RoboDK station: Config_1.rdk

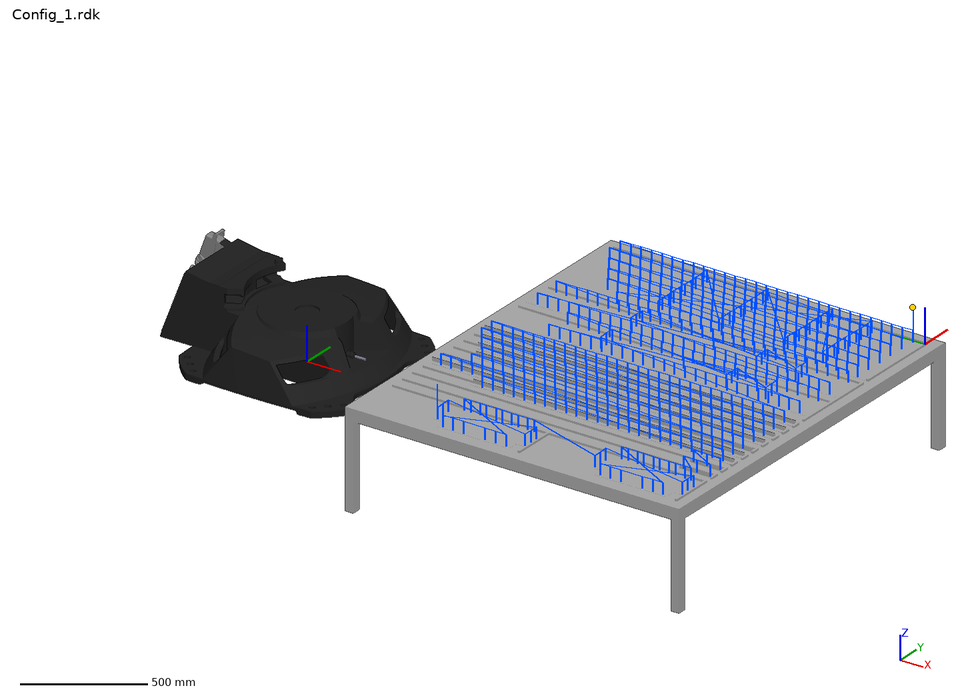
[picture v0: the station drawn from its stored meshes, robots at their saved joint values, targets as dots, program paths as lines]
Station Config_1 (saved by RoboDK 5.2.3). Poses are relative to the parent item; angles as X-Y-Z fixed-axis rotations.
  - frame KUKA KR 210 R2700 extra Base at (0, 0, 0) mm
    - robot KUKA KR 210 R2700 extra: 6 axes, payload 210 kg, reach 2696 mm, repeatability 0.06 mm, weight 1068 kg
        joint limits [-185, -140, -120, -350, -125, -350] to [185, -5, 155, 350, 125, 350]; home [0, -90, 90, 0, 0, 0]; saved at [44.26, -78.74, 122.767, 234.505, 59.006, -215.831]
      - tool Spindle, TCP at (278.6, 0, 88) mm, rotated rx 0 ry 90 rz 0 deg, size 85 x 346.5 x 128 mm
  - frame Corner First Plate at (2495, 660, 510.8) mm, rotated rx 0 ry 0 rz 90 deg
  - object Table 1 at (1700, -800, 455) mm, rotated rx 0 ry 0 rz 90 deg, size 1820 x 1600 x 475 mm, geometry from Table 1.stl
  - object Config_1 at (2495, 660, 510.8) mm, rotated rx 0 ry 0 rz 90 deg
  - machining project Path1 settings: rotZ(0) | rotX(0)*rotY(0) | rotz(0) | onStart | onPathStart | onApproach | onPoint | onRetract | onFinish | SetRPM(%1) | SetTool(%1) | Extruder(%1) | default | default | OutOnMov(%1) | OutOffMov(%1) | onPathFinish | M_RunCode(%1)
  - program Path1 (1740 instructions, listed below)
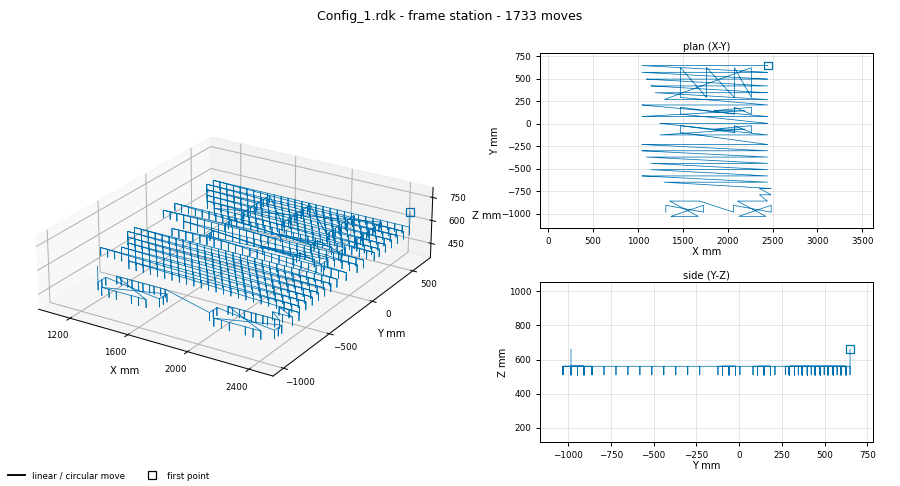
[picture p0: tool path of Config_1.rdk in frame station, 1733 of 1733 moves have a stored position in this frame; points joined in program order, loops and branches not executed]

--- program Path1 (robot KUKA KR 210 R2700 extra) ---
  Smooth(1)
  Set speed (1000.0 mm/s)
  Set Ref.: Corner First Plate
  Set Tool: Spindle
  Show Spindle
  MoveJ 1 to (-10.8, 50, 150) mm, rotated rx 180 ry 0 rz 90 deg; joints [-16.861, -44.669, 69.656, 144.341, 29.838, -148.103]
  MoveL 2 to (-10.8, 50, 150) mm, rotated rx 180 ry 0 rz 90 deg; joints [-16.861, -44.669, 69.656, 144.341, 29.838, -148.103]
  MoveL 3 to (-10.8, 50, 50) mm, rotated rx 180 ry 0 rz 90 deg; joints [-16.861, -42.157, 70.591, 147.522, 32.695, -151.823]
  MoveL 4 to (-10.8, 50, 50) mm, rotated rx 180 ry 0 rz 90 deg; joints [-16.861, -42.157, 70.591, 147.522, 32.695, -151.823]
  Set speed (150.0 mm/s)
  MoveL 5 to (-10.8, 50, -0.5) mm, rotated rx -180 ry 0 rz 90 deg; joints [-16.861, -40.791, 70.897, 148.859, 34.116, -153.424]
  MoveL 6 to (-10.8, 50, 50) mm, rotated rx 180 ry 0 rz 90 deg; joints [-16.861, -42.157, 70.591, 147.522, 32.695, -151.823]
  MoveL 7 to (-10.8, 100, 50) mm, rotated rx -180 ry 0 rz 90 deg; joints [-17.24, -44.27, 74.43, 148.298, 34.333, -152.976]
  MoveL 8 to (-10.8, 100, -0.5) mm, rotated rx -180 ry 0 rz 90 deg; joints [-17.24, -42.862, 74.73, 149.554, 35.795, -154.51]
  MoveL 9 to (-10.8, 100, 50) mm, rotated rx -180 ry 0 rz 90 deg; joints [-17.24, -44.27, 74.43, 148.298, 34.333, -152.976]
  MoveL 10 to (-10.8, 150, 50) mm, rotated rx -180 ry 0 rz 90 deg; joints [-17.637, -46.308, 78.104, 148.894, 35.906, -153.954]
  MoveL 11 to (-10.8, 150, -0.5) mm, rotated rx 180 ry 0 rz 90 deg; joints [-17.637, -44.857, 78.4, 150.085, 37.411, -155.439]
  MoveL 12 to (-10.8, 150, 50) mm, rotated rx -180 ry 0 rz 90 deg; joints [-17.637, -46.308, 78.104, 148.894, 35.906, -153.954]
  MoveL 13 to (-10.8, 200, 50) mm, rotated rx 180 ry 0 rz 90 deg; joints [-18.051, -48.282, 81.634, 149.341, 37.421, -154.79]
  MoveL 14 to (-10.8, 200, -0.5) mm, rotated rx -180 ry 0 rz 90 deg; joints [-18.051, -46.786, 81.927, 150.481, 38.968, -156.24]
  MoveL 15 to (-10.8, 200, 50) mm, rotated rx 180 ry 0 rz 90 deg; joints [-18.051, -48.282, 81.634, 149.341, 37.421, -154.79]
  MoveL 16 to (-10.8, 250, 50) mm, rotated rx 180 ry 0 rz 90 deg; joints [-18.485, -50.201, 85.037, 149.663, 38.882, -155.508]
  MoveL 17 to (-10.8, 250, -0.5) mm, rotated rx -180 ry 0 rz 90 deg; joints [-18.485, -48.66, 85.329, 150.761, 40.473, -156.934]
  MoveL 18 to (-10.8, 250, 50) mm, rotated rx 180 ry 0 rz 90 deg; joints [-18.485, -50.201, 85.037, 149.663, 38.882, -155.508]
  MoveL 19 to (-10.8, 300, 50) mm, rotated rx -180 ry 0 rz 90 deg; joints [-18.939, -52.073, 88.328, 149.877, 40.293, -156.128]
  MoveL 20 to (-10.8, 300, -0.5) mm, rotated rx 180 ry 0 rz 90 deg; joints [-18.939, -50.484, 88.62, 150.941, 41.929, -157.54]
  MoveL 21 to (-10.8, 300, 50) mm, rotated rx -180 ry 0 rz 90 deg; joints [-18.939, -52.073, 88.328, 149.877, 40.293, -156.128]
  MoveL 22 to (-10.8, 350, 50) mm, rotated rx 180 ry 0 rz 90 deg; joints [-19.415, -53.906, 91.518, 149.994, 41.659, -156.663]
  MoveL 23 to (-10.8, 350, -0.5) mm, rotated rx 180 ry 0 rz 90 deg; joints [-19.415, -52.267, 91.81, 151.032, 43.339, -158.069]
  MoveL 24 to (-10.8, 350, 50) mm, rotated rx 180 ry 0 rz 90 deg; joints [-19.415, -53.906, 91.518, 149.994, 41.659, -156.663]
  MoveL 25 to (-10.8, 400, 50) mm, rotated rx 180 ry 0 rz 90 deg; joints [-19.914, -55.704, 94.616, 150.026, 42.981, -157.123]
  MoveL 26 to (-10.8, 400, -0.5) mm, rotated rx -180 ry 0 rz 90 deg; joints [-19.914, -54.013, 94.91, 151.042, 44.709, -158.532]
  MoveL 27 to (-10.8, 400, 50) mm, rotated rx 180 ry 0 rz 90 deg; joints [-19.914, -55.704, 94.616, 150.026, 42.981, -157.123]
  MoveL 28 to (-10.8, 450, 50) mm, rotated rx 180 ry 0 rz 90 deg; joints [-20.439, -57.473, 97.631, 149.977, 44.262, -157.517]
  MoveL 29 to (-10.8, 450, -0.5) mm, rotated rx 180 ry 0 rz 90 deg; joints [-20.439, -55.727, 97.926, 150.978, 46.038, -158.936]
  MoveL 30 to (-10.8, 450, 50) mm, rotated rx 180 ry 0 rz 90 deg; joints [-20.439, -57.473, 97.631, 149.977, 44.262, -157.517]
  MoveL 31 to (-10.8, 500, 50) mm, rotated rx -180 ry 0 rz 90 deg; joints [-20.991, -59.217, 100.569, 149.854, 45.504, -157.852]
  MoveL 32 to (-10.8, 500, -0.5) mm, rotated rx 180 ry 0 rz 90 deg; joints [-20.991, -57.414, 100.867, 150.844, 47.331, -159.288]
  MoveL 33 to (-10.8, 500, 50) mm, rotated rx -180 ry 0 rz 90 deg; joints [-20.991, -59.217, 100.569, 149.854, 45.504, -157.852]
  MoveL 34 to (-10.8, 550, 50) mm, rotated rx 180 ry 0 rz 90 deg; joints [-21.572, -60.942, 103.435, 149.66, 46.709, -158.133]
  MoveL 35 to (-10.8, 550, -0.5) mm, rotated rx 180 ry 0 rz 90 deg; joints [-21.572, -59.078, 103.738, 150.643, 48.588, -159.592]
  MoveL 36 to (-10.8, 550, 50) mm, rotated rx 180 ry 0 rz 90 deg; joints [-21.572, -60.942, 103.435, 149.66, 46.709, -158.133]
  MoveL 37 to (-10.8, 600, 50) mm, rotated rx 180 ry 0 rz 90 deg; joints [-22.185, -62.649, 106.236, 149.397, 47.878, -158.362]
  MoveL 38 to (-10.8, 600, -0.5) mm, rotated rx 180 ry 0 rz 90 deg; joints [-22.185, -60.721, 106.543, 150.377, 49.812, -159.851]
  MoveL 39 to (-10.8, 600, 50) mm, rotated rx 180 ry 0 rz 90 deg; joints [-22.185, -62.649, 106.236, 149.397, 47.878, -158.362]
  MoveL 40 to (-10.8, 650, 50) mm, rotated rx 180 ry 0 rz 90 deg; joints [-22.832, -64.344, 108.975, 149.067, 49.013, -158.542]
  MoveL 41 to (-10.8, 650, -0.5) mm, rotated rx 180 ry 0 rz 90 deg; joints [-22.832, -62.348, 109.287, 150.048, 51.003, -160.069]
  MoveL 42 to (-10.8, 650, 50) mm, rotated rx 180 ry 0 rz 90 deg; joints [-22.832, -64.344, 108.975, 149.067, 49.013, -158.542]
  MoveL 43 to (-10.8, 700, 50) mm, rotated rx -180 ry 0 rz 90 deg; joints [-23.515, -66.029, 111.655, 148.669, 50.113, -158.676]
  MoveL 44 to (-10.8, 700, -0.5) mm, rotated rx 180 ry 0 rz 90 deg; joints [-23.515, -63.961, 111.973, 149.655, 52.163, -160.247]
  MoveL 45 to (-10.8, 700, 50) mm, rotated rx -180 ry 0 rz 90 deg; joints [-23.515, -66.029, 111.655, 148.669, 50.113, -158.676]
  MoveL 46 to (-10.8, 750, 50) mm, rotated rx 180 ry 0 rz 90 deg; joints [-24.238, -67.708, 114.279, 148.204, 51.181, -158.763]
  MoveL 47 to (-10.8, 750, -0.5) mm, rotated rx 180 ry 0 rz 90 deg; joints [-24.238, -65.564, 114.604, 149.198, 53.292, -160.386]
  MoveL 48 to (-10.8, 750, 50) mm, rotated rx 180 ry 0 rz 90 deg; joints [-24.238, -67.708, 114.279, 148.204, 51.181, -158.763]
  MoveL 49 to (-10.8, 800, 50) mm, rotated rx -180 ry 0 rz 90 deg; joints [-25.003, -69.384, 116.85, 147.669, 52.216, -158.805]
  MoveL 50 to (-10.8, 800, -0.5) mm, rotated rx 180 ry 0 rz 90 deg; joints [-25.003, -67.159, 117.183, 148.675, 54.391, -160.488]
  MoveL 51 to (-10.8, 800, 50) mm, rotated rx -180 ry 0 rz 90 deg; joints [-25.003, -69.384, 116.85, 147.669, 52.216, -158.805]
  MoveL 52 to (-10.8, 850, 50) mm, rotated rx -180 ry 0 rz 90 deg; joints [-25.816, -71.061, 119.369, 147.064, 53.22, -158.799]
  MoveL 53 to (-10.8, 850, -0.5) mm, rotated rx 180 ry 0 rz 90 deg; joints [-25.816, -68.749, 119.711, 148.085, 55.46, -160.551]
  MoveL 54 to (-10.8, 850, 50) mm, rotated rx -180 ry 0 rz 90 deg; joints [-25.816, -71.061, 119.369, 147.064, 53.22, -158.799]
  MoveL 55 to (-10.8, 900, 50) mm, rotated rx 180 ry 0 rz 90 deg; joints [-26.678, -72.742, 121.838, 146.383, 54.192, -158.746]
  MoveL 56 to (-10.8, 900, -0.5) mm, rotated rx -180 ry 0 rz 90 deg; joints [-26.678, -70.337, 122.19, 147.424, 56.501, -160.575]
  MoveL 57 to (-10.8, 900, 50) mm, rotated rx 180 ry 0 rz 90 deg; joints [-26.678, -72.742, 121.838, 146.383, 54.192, -158.746]
  MoveL 58 to (-10.8, 950, 50) mm, rotated rx -180 ry 0 rz 90 deg; joints [-27.596, -74.43, 124.259, 145.626, 55.132, -158.641]
  MoveL 59 to (-10.8, 950, -0.5) mm, rotated rx -180 ry 0 rz 90 deg; joints [-27.596, -71.926, 124.621, 146.689, 57.513, -160.559]
  MoveL 60 to (-10.8, 950, 50) mm, rotated rx -180 ry 0 rz 90 deg; joints [-27.596, -74.43, 124.259, 145.626, 55.132, -158.641]
  MoveL 61 to (-10.8, 1000, 50) mm, rotated rx 180 ry 0 rz 90 deg; joints [-28.574, -76.128, 126.631, 144.786, 56.043, -158.484]
  MoveL 62 to (-10.8, 1000, -0.5) mm, rotated rx 180 ry 0 rz 90 deg; joints [-28.574, -73.519, 127.005, 145.877, 58.497, -160.501]
  MoveL 63 to (-10.8, 1000, 50) mm, rotated rx 180 ry 0 rz 90 deg; joints [-28.574, -76.128, 126.631, 144.786, 56.043, -158.484]
  MoveL 64 to (-10.8, 1050, 50) mm, rotated rx -180 ry 0 rz 90 deg; joints [-29.617, -77.842, 128.955, 143.858, 56.923, -158.269]
  MoveL 65 to (-10.8, 1050, -0.5) mm, rotated rx 180 ry 0 rz 90 deg; joints [-29.617, -75.119, 129.342, 144.981, 59.453, -160.398]
  MoveL 66 to (-10.8, 1050, 50) mm, rotated rx -180 ry 0 rz 90 deg; joints [-29.617, -77.842, 128.955, 143.858, 56.923, -158.269]
  MoveL 67 to (-10.8, 1100, 50) mm, rotated rx 180 ry 0 rz 90 deg; joints [-30.732, -79.573, 131.231, 142.838, 57.775, -157.992]
  MoveL 68 to (-10.8, 1100, -0.5) mm, rotated rx -180 ry 0 rz 90 deg; joints [-30.732, -76.729, 131.632, 143.997, 60.382, -160.246]
  MoveL 69 to (-10.8, 1100, 50) mm, rotated rx 180 ry 0 rz 90 deg; joints [-30.732, -79.573, 131.231, 142.838, 57.775, -157.992]
  MoveL 70 to (-10.8, 1150, 50) mm, rotated rx 180 ry 0 rz 90 deg; joints [-31.924, -81.327, 133.457, 141.718, 58.599, -157.647]
  MoveL 71 to (-10.8, 1150, -0.5) mm, rotated rx 180 ry 0 rz 90 deg; joints [-31.924, -78.352, 133.874, 142.918, 61.284, -160.042]
  MoveL 72 to (-10.8, 1150, 50) mm, rotated rx 180 ry 0 rz 90 deg; joints [-31.924, -81.327, 133.457, 141.718, 58.599, -157.647]
  MoveL 73 to (-10.8, 1200, 50) mm, rotated rx 180 ry 0 rz 90 deg; joints [-33.202, -83.108, 135.634, 140.49, 59.397, -157.227]
  MoveL 74 to (-10.8, 1200, -0.5) mm, rotated rx 180 ry 0 rz 90 deg; joints [-33.202, -79.993, 136.068, 141.737, 62.161, -159.78]
  MoveL 75 to (-10.8, 1200, 50) mm, rotated rx 180 ry 0 rz 90 deg; joints [-33.202, -83.108, 135.634, 140.49, 59.397, -157.227]
  MoveL 76 to (-10.8, 1250, 50) mm, rotated rx -180 ry 0 rz 90 deg; joints [-34.574, -84.92, 137.758, 139.147, 60.172, -156.726]
  MoveL 77 to (-10.8, 1250, -0.5) mm, rotated rx -180 ry 0 rz 90 deg; joints [-34.574, -81.654, 138.211, 140.446, 63.014, -159.455]
  MoveL 78 to (-10.8, 1250, 50) mm, rotated rx -180 ry 0 rz 90 deg; joints [-34.574, -84.92, 137.758, 139.147, 60.172, -156.726]
  MoveL 79 to (-10.8, 1300, 50) mm, rotated rx 180 ry 0 rz 90 deg; joints [-36.047, -86.767, 139.828, 137.68, 60.929, -156.133]
  MoveL 80 to (-10.8, 1300, -0.5) mm, rotated rx 180 ry 0 rz 90 deg; joints [-36.047, -83.339, 140.302, 139.037, 63.846, -159.059]
  MoveL 81 to (-10.8, 1300, 50) mm, rotated rx 180 ry 0 rz 90 deg; joints [-36.047, -86.767, 139.828, 137.68, 60.929, -156.133]
  MoveL 82 to (-10.8, 1350, 50) mm, rotated rx 180 ry 0 rz 90 deg; joints [-37.633, -88.655, 141.842, 136.078, 61.671, -155.439]
  MoveL 83 to (-10.8, 1350, -0.5) mm, rotated rx 180 ry 0 rz 90 deg; joints [-37.633, -85.052, 142.339, 137.499, 64.659, -158.585]
  MoveL 84 to (-10.8, 1350, 50) mm, rotated rx 180 ry 0 rz 90 deg; joints [-37.633, -88.655, 141.842, 136.078, 61.671, -155.439]
  MoveL 85 to (-10.8, 1400, 50) mm, rotated rx -180 ry 0 rz 90 deg; joints [-39.341, -90.587, 143.795, 134.333, 62.407, -154.634]
  MoveL 86 to (-10.8, 1400, -0.5) mm, rotated rx 180 ry 0 rz 90 deg; joints [-39.341, -86.798, 144.317, 135.822, 65.461, -158.023]
  MoveL 87 to (-10.8, 1400, 50) mm, rotated rx -180 ry 0 rz 90 deg; joints [-39.341, -90.587, 143.795, 134.333, 62.407, -154.634]
  MoveL 88 to (-10.8, 1450, 50) mm, rotated rx 180 ry 0 rz 90 deg; joints [-41.184, -92.567, 145.684, 132.434, 63.147, -153.707]
  MoveL 89 to (-10.8, 1450, -0.5) mm, rotated rx -180 ry 0 rz 90 deg; joints [-41.184, -88.578, 146.233, 133.998, 66.256, -157.364]
  MoveL 90 to (-10.8, 1450, 50) mm, rotated rx 180 ry 0 rz 90 deg; joints [-41.184, -92.567, 145.684, 132.434, 63.147, -153.707]
  MoveL 91 to (-86.48, 50, 50) mm, rotated rx -180 ry 0 rz 90 deg; joints [-14.989, -43.085, 72.28, 151.237, 32.514, -155.162]
  MoveL 92 to (-86.48, 50, -0.5) mm, rotated rx -180 ry 0 rz 90 deg; joints [-14.989, -41.7, 72.583, 152.451, 34.002, -156.614]
  MoveL 93 to (-86.48, 50, 50) mm, rotated rx -180 ry 0 rz 90 deg; joints [-14.989, -43.085, 72.28, 151.237, 32.514, -155.162]
  MoveL 94 to (-86.48, 100, 50) mm, rotated rx 180 ry 0 rz 90 deg; joints [-15.331, -45.185, 76.083, 151.903, 34.152, -156.164]
  MoveL 95 to (-86.48, 100, -0.5) mm, rotated rx -180 ry 0 rz 90 deg; joints [-15.331, -43.758, 76.381, 153.045, 35.682, -157.556]
  MoveL 96 to (-86.48, 100, 50) mm, rotated rx 180 ry 0 rz 90 deg; joints [-15.331, -45.185, 76.083, 151.903, 34.152, -156.164]
  MoveL 97 to (-86.48, 150, 50) mm, rotated rx 180 ry 0 rz 90 deg; joints [-15.688, -47.215, 79.729, 152.412, 35.724, -157.013]
  MoveL 98 to (-86.48, 150, -0.5) mm, rotated rx 180 ry 0 rz 90 deg; joints [-15.688, -45.744, 80.024, 153.496, 37.296, -158.362]
  MoveL 99 to (-86.48, 150, 50) mm, rotated rx 180 ry 0 rz 90 deg; joints [-15.688, -47.215, 79.729, 152.412, 35.724, -157.013]
  MoveL 100 to (-86.48, 200, 50) mm, rotated rx -180 ry 0 rz 90 deg; joints [-16.062, -49.185, 83.239, 152.79, 37.234, -157.738]
  MoveL 101 to (-86.48, 200, -0.5) mm, rotated rx 180 ry 0 rz 90 deg; joints [-16.062, -47.668, 83.531, 153.829, 38.851, -159.057]
  MoveL 102 to (-86.48, 200, 50) mm, rotated rx -180 ry 0 rz 90 deg; joints [-16.062, -49.185, 83.239, 152.79, 37.234, -157.738]
  MoveL 103 to (-86.48, 250, 50) mm, rotated rx 180 ry 0 rz 90 deg; joints [-16.453, -51.104, 86.628, 153.058, 38.69, -158.361]
  MoveL 104 to (-86.48, 250, -0.5) mm, rotated rx 180 ry 0 rz 90 deg; joints [-16.453, -49.54, 86.92, 154.059, 40.351, -159.659]
  MoveL 105 to (-86.48, 250, 50) mm, rotated rx 180 ry 0 rz 90 deg; joints [-16.453, -51.104, 86.628, 153.058, 38.69, -158.361]
  MoveL 106 to (-86.48, 300, 50) mm, rotated rx -180 ry 0 rz 90 deg; joints [-16.864, -52.98, 89.91, 153.229, 40.094, -158.896]
  MoveL 107 to (-86.48, 300, -0.5) mm, rotated rx 180 ry 0 rz 90 deg; joints [-16.864, -51.367, 90.202, 154.201, 41.802, -160.183]
  MoveL 108 to (-86.48, 300, 50) mm, rotated rx -180 ry 0 rz 90 deg; joints [-16.864, -52.98, 89.91, 153.229, 40.094, -158.896]
  MoveL 109 to (-86.48, 350, 50) mm, rotated rx 180 ry 0 rz 90 deg; joints [-17.294, -54.819, 93.096, 153.315, 41.45, -159.357]
  MoveL 110 to (-86.48, 350, -0.5) mm, rotated rx 180 ry 0 rz 90 deg; joints [-17.294, -53.155, 93.389, 154.264, 43.206, -160.641]
  MoveL 111 to (-86.48, 350, 50) mm, rotated rx 180 ry 0 rz 90 deg; joints [-17.294, -54.819, 93.096, 153.315, 41.45, -159.357]
  MoveL 112 to (-86.48, 400, 50) mm, rotated rx 180 ry 0 rz 90 deg; joints [-17.747, -56.627, 96.194, 153.323, 42.76, -159.751]
  MoveL 113 to (-86.48, 400, -0.5) mm, rotated rx -180 ry 0 rz 90 deg; joints [-17.747, -54.909, 96.489, 154.255, 44.567, -161.039]
  MoveL 114 to (-86.48, 400, 50) mm, rotated rx 180 ry 0 rz 90 deg; joints [-17.747, -56.627, 96.194, 153.323, 42.76, -159.751]
  MoveL 115 to (-86.48, 450, 50) mm, rotated rx 180 ry 0 rz 90 deg; joints [-18.223, -58.41, 99.213, 153.26, 44.028, -160.087]
  MoveL 116 to (-86.48, 450, -0.5) mm, rotated rx -180 ry 0 rz 90 deg; joints [-18.223, -56.634, 99.51, 154.179, 45.887, -161.386]
  MoveL 117 to (-86.48, 450, 50) mm, rotated rx 180 ry 0 rz 90 deg; joints [-18.223, -58.41, 99.213, 153.26, 44.028, -160.087]
  MoveL 118 to (-86.48, 500, 50) mm, rotated rx 180 ry 0 rz 90 deg; joints [-18.725, -60.17, 102.158, 153.129, 45.255, -160.369]
  MoveL 119 to (-86.48, 500, -0.5) mm, rotated rx 180 ry 0 rz 90 deg; joints [-18.725, -58.334, 102.459, 154.04, 47.169, -161.686]
  MoveL 120 to (-86.48, 500, 50) mm, rotated rx 180 ry 0 rz 90 deg; joints [-18.725, -60.17, 102.158, 153.129, 45.255, -160.369]
  MoveL 121 to (-86.48, 550, 50) mm, rotated rx 180 ry 0 rz 90 deg; joints [-19.253, -61.914, 105.035, 152.934, 46.442, -160.602]
  MoveL 122 to (-86.48, 550, -0.5) mm, rotated rx 180 ry 0 rz 90 deg; joints [-19.253, -60.014, 105.341, 153.841, 48.414, -161.943]
  MoveL 123 to (-86.48, 550, 50) mm, rotated rx 180 ry 0 rz 90 deg; joints [-19.253, -61.914, 105.035, 152.934, 46.442, -160.602]
  MoveL 124 to (-86.48, 600, 50) mm, rotated rx 180 ry 0 rz 90 deg; joints [-19.812, -63.645, 107.85, 152.675, 47.591, -160.788]
  MoveL 125 to (-86.48, 600, -0.5) mm, rotated rx 180 ry 0 rz 90 deg; joints [-19.812, -61.677, 108.16, 153.583, 49.623, -162.161]
  MoveL 126 to (-86.48, 600, 50) mm, rotated rx 180 ry 0 rz 90 deg; joints [-19.812, -63.645, 107.85, 152.675, 47.591, -160.788]
  MoveL 127 to (-86.48, 650, 50) mm, rotated rx 180 ry 0 rz 90 deg; joints [-20.402, -65.366, 110.606, 152.354, 48.702, -160.93]
  MoveL 128 to (-86.48, 650, -0.5) mm, rotated rx 180 ry 0 rz 90 deg; joints [-20.402, -63.327, 110.922, 153.265, 50.797, -162.34]
  MoveL 129 to (-86.48, 650, 50) mm, rotated rx 180 ry 0 rz 90 deg; joints [-20.402, -65.366, 110.606, 152.354, 48.702, -160.93]
  MoveL 130 to (-86.48, 700, 50) mm, rotated rx -180 ry 0 rz 90 deg; joints [-21.027, -67.082, 113.306, 151.97, 49.776, -161.027]
  MoveL 131 to (-86.48, 700, -0.5) mm, rotated rx -180 ry 0 rz 90 deg; joints [-21.027, -64.967, 113.629, 152.889, 51.938, -162.482]
  MoveL 132 to (-86.48, 700, 50) mm, rotated rx -180 ry 0 rz 90 deg; joints [-21.027, -67.082, 113.306, 151.97, 49.776, -161.027]
  MoveL 133 to (-86.48, 750, 50) mm, rotated rx -180 ry 0 rz 90 deg; joints [-21.689, -68.796, 115.953, 151.523, 50.813, -161.081]
  MoveL 134 to (-86.48, 750, -0.5) mm, rotated rx 180 ry 0 rz 90 deg; joints [-21.689, -66.6, 116.284, 152.453, 53.044, -162.589]
  MoveL 135 to (-86.48, 750, 50) mm, rotated rx -180 ry 0 rz 90 deg; joints [-21.689, -68.796, 115.953, 151.523, 50.813, -161.081]
  MoveL 136 to (-86.48, 800, 50) mm, rotated rx -180 ry 0 rz 90 deg; joints [-22.392, -70.512, 118.55, 151.01, 51.814, -161.091]
  MoveL 137 to (-86.48, 800, -0.5) mm, rotated rx 180 ry 0 rz 90 deg; joints [-22.392, -68.229, 118.89, 151.955, 54.118, -162.66]
  MoveL 138 to (-86.48, 800, 50) mm, rotated rx -180 ry 0 rz 90 deg; joints [-22.392, -70.512, 118.55, 151.01, 51.814, -161.091]
  MoveL 139 to (-86.48, 850, 50) mm, rotated rx -180 ry 0 rz 90 deg; joints [-23.14, -72.235, 121.099, 150.428, 52.777, -161.056]
  MoveL 140 to (-86.48, 850, -0.5) mm, rotated rx 180 ry 0 rz 90 deg; joints [-23.14, -69.858, 121.448, 151.392, 55.159, -162.694]
  MoveL 141 to (-86.48, 850, 50) mm, rotated rx -180 ry 0 rz 90 deg; joints [-23.14, -72.235, 121.099, 150.428, 52.777, -161.056]
  MoveL 142 to (-86.48, 900, 50) mm, rotated rx 180 ry 0 rz 90 deg; joints [-23.936, -73.967, 123.602, 149.775, 53.704, -160.972]
  MoveL 143 to (-86.48, 900, -0.5) mm, rotated rx 180 ry 0 rz 90 deg; joints [-23.936, -71.491, 123.961, 150.762, 56.166, -162.69]
  MoveL 144 to (-86.48, 900, 50) mm, rotated rx 180 ry 0 rz 90 deg; joints [-23.936, -73.967, 123.602, 149.775, 53.704, -160.972]
  MoveL 145 to (-86.48, 950, 50) mm, rotated rx -180 ry 0 rz 90 deg; joints [-24.786, -75.714, 126.058, 149.045, 54.593, -160.837]
  MoveL 146 to (-86.48, 950, -0.5) mm, rotated rx 180 ry 0 rz 90 deg; joints [-24.786, -73.131, 126.429, 150.06, 57.14, -162.646]
  MoveL 147 to (-86.48, 950, 50) mm, rotated rx -180 ry 0 rz 90 deg; joints [-24.786, -75.714, 126.058, 149.045, 54.593, -160.837]
  MoveL 148 to (-86.48, 1000, 50) mm, rotated rx 180 ry 0 rz 90 deg; joints [-25.694, -77.479, 128.47, 148.234, 55.444, -160.648]
  MoveL 149 to (-86.48, 1000, -0.5) mm, rotated rx 180 ry 0 rz 90 deg; joints [-25.694, -74.781, 128.854, 149.282, 58.079, -162.559]
  MoveL 150 to (-86.48, 1000, 50) mm, rotated rx 180 ry 0 rz 90 deg; joints [-25.694, -77.479, 128.47, 148.234, 55.444, -160.648]
  MoveL 151 to (-86.48, 1050, 50) mm, rotated rx 180 ry 0 rz 90 deg; joints [-26.666, -79.269, 130.836, 147.336, 56.256, -160.398]
  MoveL 152 to (-86.48, 1050, -0.5) mm, rotated rx -180 ry 0 rz 90 deg; joints [-26.666, -76.447, 131.235, 148.422, 58.985, -162.426]
  MoveL 153 to (-86.48, 1050, 50) mm, rotated rx 180 ry 0 rz 90 deg; joints [-26.666, -79.269, 130.836, 147.336, 56.256, -160.398]
  MoveL 154 to (-86.48, 1100, 50) mm, rotated rx 180 ry 0 rz 90 deg; joints [-27.709, -81.088, 133.158, 146.342, 57.029, -160.081]
  MoveL 155 to (-86.48, 1100, -0.5) mm, rotated rx 180 ry 0 rz 90 deg; joints [-27.709, -78.131, 133.573, 147.473, 59.855, -162.242]
  MoveL 156 to (-86.48, 1100, 50) mm, rotated rx 180 ry 0 rz 90 deg; joints [-27.709, -81.088, 133.158, 146.342, 57.029, -160.081]
  MoveL 157 to (-86.48, 1150, 50) mm, rotated rx 180 ry 0 rz 90 deg; joints [-28.829, -82.943, 135.435, 145.246, 57.764, -159.69]
  MoveL 158 to (-86.48, 1150, -0.5) mm, rotated rx 180 ry 0 rz 90 deg; joints [-28.829, -79.841, 135.868, 146.428, 60.689, -162]
  MoveL 159 to (-86.48, 1150, 50) mm, rotated rx 180 ry 0 rz 90 deg; joints [-28.829, -82.943, 135.435, 145.246, 57.764, -159.69]
  MoveL 160 to (-86.48, 1200, 50) mm, rotated rx 180 ry 0 rz 90 deg; joints [-30.034, -84.839, 137.665, 144.036, 58.459, -159.215]
  MoveL 161 to (-86.48, 1200, -0.5) mm, rotated rx -180 ry 0 rz 90 deg; joints [-30.034, -81.58, 138.118, 145.278, 61.487, -161.695]
  MoveL 162 to (-86.48, 1200, 50) mm, rotated rx 180 ry 0 rz 90 deg; joints [-30.034, -84.839, 137.665, 144.036, 58.459, -159.215]
  MoveL 163 to (-86.48, 1250, 50) mm, rotated rx -180 ry 0 rz 90 deg; joints [-31.334, -86.785, 139.848, 142.703, 59.117, -158.645]
  MoveL 164 to (-86.48, 1250, -0.5) mm, rotated rx 180 ry 0 rz 90 deg; joints [-31.334, -83.355, 140.322, 144.012, 62.25, -161.317]
  MoveL 165 to (-86.48, 1250, 50) mm, rotated rx -180 ry 0 rz 90 deg; joints [-31.334, -86.785, 139.848, 142.703, 59.117, -158.645]
  MoveL 166 to (-86.48, 1300, 50) mm, rotated rx -180 ry 0 rz 90 deg; joints [-32.739, -88.788, 141.98, 141.234, 59.738, -157.967]
  MoveL 167 to (-86.48, 1300, -0.5) mm, rotated rx -180 ry 0 rz 90 deg; joints [-32.739, -85.173, 142.478, 142.62, 62.977, -160.857]
  MoveL 168 to (-86.48, 1300, 50) mm, rotated rx -180 ry 0 rz 90 deg; joints [-32.739, -88.788, 141.98, 141.234, 59.738, -157.967]
  MoveL 169 to (-86.48, 1350, 50) mm, rotated rx 180 ry 0 rz 90 deg; joints [-34.26, -90.856, 144.059, 139.615, 60.327, -157.164]
  MoveL 170 to (-86.48, 1350, -0.5) mm, rotated rx -180 ry 0 rz 90 deg; joints [-34.26, -87.04, 144.584, 141.089, 63.67, -160.301]
  MoveL 171 to (-86.48, 1350, 50) mm, rotated rx 180 ry 0 rz 90 deg; joints [-34.26, -90.856, 144.059, 139.615, 60.327, -157.164]
  MoveL 172 to (-86.48, 1400, 50) mm, rotated rx -180 ry 0 rz 90 deg; joints [-35.91, -92.999, 146.082, 137.831, 60.889, -156.219]
  MoveL 173 to (-86.48, 1400, -0.5) mm, rotated rx -180 ry 0 rz 90 deg; joints [-35.91, -88.966, 146.637, 139.404, 64.333, -159.635]
  MoveL 174 to (-86.48, 1400, 50) mm, rotated rx -180 ry 0 rz 90 deg; joints [-35.91, -92.999, 146.082, 137.831, 60.889, -156.219]
  MoveL 175 to (-86.48, 1450, 50) mm, rotated rx 180 ry 0 rz 90 deg; joints [-37.702, -95.228, 148.043, 135.867, 61.433, -155.112]
  MoveL 176 to (-86.48, 1450, -0.5) mm, rotated rx 180 ry 0 rz 90 deg; joints [-37.702, -90.959, 148.632, 137.551, 64.97, -158.843]
  MoveL 177 to (-86.48, 1450, 50) mm, rotated rx 180 ry 0 rz 90 deg; joints [-37.702, -95.228, 148.043, 135.867, 61.433, -155.112]
  MoveL 178 to (-162.16, 50, 50) mm, rotated rx 180 ry 0 rz 90 deg; joints [-13.084, -43.892, 73.746, 154.972, 32.351, -158.474]
  MoveL 179 to (-162.16, 50, -0.5) mm, rotated rx 180 ry 0 rz 90 deg; joints [-13.084, -42.492, 74.047, 156.053, 33.899, -159.764]
  MoveL 180 to (-162.16, 50, 50) mm, rotated rx 180 ry 0 rz 90 deg; joints [-13.084, -43.892, 73.746, 154.972, 32.351, -158.474]
  MoveL 181 to (-162.16, 100, 50) mm, rotated rx 180 ry 0 rz 90 deg; joints [-13.386, -45.983, 77.52, 155.536, 33.989, -159.332]
  MoveL 182 to (-162.16, 100, -0.5) mm, rotated rx 180 ry 0 rz 90 deg; joints [-13.386, -44.539, 77.816, 156.553, 35.579, -160.57]
  MoveL 183 to (-162.16, 100, 50) mm, rotated rx 180 ry 0 rz 90 deg; joints [-13.386, -45.983, 77.52, 155.536, 33.989, -159.332]
  MoveL 184 to (-162.16, 150, 50) mm, rotated rx -180 ry 0 rz 90 deg; joints [-13.701, -48.007, 81.145, 155.964, 35.558, -160.058]
  MoveL 185 to (-162.16, 150, -0.5) mm, rotated rx 180 ry 0 rz 90 deg; joints [-13.701, -46.519, 81.439, 156.931, 37.192, -161.259]
  MoveL 186 to (-162.16, 150, 50) mm, rotated rx -180 ry 0 rz 90 deg; joints [-13.701, -48.007, 81.145, 155.964, 35.558, -160.058]
  MoveL 187 to (-162.16, 200, 50) mm, rotated rx 180 ry 0 rz 90 deg; joints [-14.032, -49.975, 84.639, 156.279, 37.064, -160.678]
  MoveL 188 to (-162.16, 200, -0.5) mm, rotated rx -180 ry 0 rz 90 deg; joints [-14.032, -48.44, 84.931, 157.206, 38.743, -161.852]
  MoveL 189 to (-162.16, 200, 50) mm, rotated rx 180 ry 0 rz 90 deg; joints [-14.032, -49.975, 84.639, 156.279, 37.064, -160.678]
  MoveL 190 to (-162.16, 250, 50) mm, rotated rx 180 ry 0 rz 90 deg; joints [-14.378, -51.896, 88.018, 156.498, 38.514, -161.209]
  MoveL 191 to (-162.16, 250, -0.5) mm, rotated rx 180 ry 0 rz 90 deg; joints [-14.378, -50.312, 88.31, 157.393, 40.239, -162.366]
  MoveL 192 to (-162.16, 250, 50) mm, rotated rx 180 ry 0 rz 90 deg; joints [-14.378, -51.896, 88.018, 156.498, 38.514, -161.209]
  MoveL 193 to (-162.16, 300, 50) mm, rotated rx 180 ry 0 rz 90 deg; joints [-14.742, -53.777, 91.294, 156.633, 39.91, -161.664]
  MoveL 194 to (-162.16, 300, -0.5) mm, rotated rx 180 ry 0 rz 90 deg; joints [-14.742, -52.142, 91.587, 157.503, 41.685, -162.813]
  MoveL 195 to (-162.16, 300, 50) mm, rotated rx 180 ry 0 rz 90 deg; joints [-14.742, -53.777, 91.294, 156.633, 39.91, -161.664]
  MoveL 196 to (-162.16, 350, 50) mm, rotated rx -180 ry 0 rz 90 deg; joints [-15.124, -55.623, 94.478, 156.693, 41.256, -162.054]
  MoveL 197 to (-162.16, 350, -0.5) mm, rotated rx -180 ry 0 rz 90 deg; joints [-15.124, -53.935, 94.772, 157.544, 43.082, -163.202]
  MoveL 198 to (-162.16, 350, 50) mm, rotated rx -180 ry 0 rz 90 deg; joints [-15.124, -55.623, 94.478, 156.693, 41.256, -162.054]
  MoveL 199 to (-162.16, 400, 50) mm, rotated rx 180 ry 0 rz 90 deg; joints [-15.526, -57.442, 97.578, 156.685, 42.556, -162.387]
  MoveL 200 to (-162.16, 400, -0.5) mm, rotated rx 180 ry 0 rz 90 deg; joints [-15.526, -55.697, 97.874, 157.522, 44.436, -163.54]
  MoveL 201 to (-162.16, 400, 50) mm, rotated rx 180 ry 0 rz 90 deg; joints [-15.526, -57.442, 97.578, 156.685, 42.556, -162.387]
  MoveL 202 to (-162.16, 450, 50) mm, rotated rx -180 ry 0 rz 90 deg; joints [-15.949, -59.237, 100.601, 156.614, 43.811, -162.668]
  MoveL 203 to (-162.16, 450, -0.5) mm, rotated rx -180 ry 0 rz 90 deg; joints [-15.949, -57.433, 100.9, 157.441, 45.747, -163.833]
  MoveL 204 to (-162.16, 450, 50) mm, rotated rx -180 ry 0 rz 90 deg; joints [-15.949, -59.237, 100.601, 156.614, 43.811, -162.668]
  MoveL 205 to (-162.16, 500, 50) mm, rotated rx -180 ry 0 rz 90 deg; joints [-16.396, -61.014, 103.555, 156.482, 45.022, -162.902]
  MoveL 206 to (-162.16, 500, -0.5) mm, rotated rx 180 ry 0 rz 90 deg; joints [-16.396, -59.147, 103.858, 157.304, 47.017, -164.085]
  MoveL 207 to (-162.16, 500, 50) mm, rotated rx -180 ry 0 rz 90 deg; joints [-16.396, -61.014, 103.555, 156.482, 45.022, -162.902]
  MoveL 208 to (-162.16, 550, 50) mm, rotated rx -180 ry 0 rz 90 deg; joints [-16.867, -62.777, 106.443, 156.293, 46.192, -163.092]
  MoveL 209 to (-162.16, 550, -0.5) mm, rotated rx 180 ry 0 rz 90 deg; joints [-16.867, -60.844, 106.751, 157.113, 48.25, -164.299]
  MoveL 210 to (-162.16, 550, 50) mm, rotated rx -180 ry 0 rz 90 deg; joints [-16.867, -62.777, 106.443, 156.293, 46.192, -163.092]
  MoveL 211 to (-162.16, 600, 50) mm, rotated rx 180 ry 0 rz 90 deg; joints [-17.365, -64.529, 109.272, 156.047, 47.32, -163.24]
  MoveL 212 to (-162.16, 600, -0.5) mm, rotated rx -180 ry 0 rz 90 deg; joints [-17.365, -62.526, 109.585, 156.869, 49.444, -164.478]
  MoveL 213 to (-162.16, 600, 50) mm, rotated rx 180 ry 0 rz 90 deg; joints [-17.365, -64.529, 109.272, 156.047, 47.32, -163.24]
  MoveL 214 to (-162.16, 650, 50) mm, rotated rx 180 ry 0 rz 90 deg; joints [-17.893, -66.277, 112.044, 155.744, 48.408, -163.347]
  MoveL 215 to (-162.16, 650, -0.5) mm, rotated rx 180 ry 0 rz 90 deg; joints [-17.893, -64.198, 112.364, 156.572, 50.601, -164.622]
  MoveL 216 to (-162.16, 650, 50) mm, rotated rx 180 ry 0 rz 90 deg; joints [-17.893, -66.277, 112.044, 155.744, 48.408, -163.347]
  MoveL 217 to (-162.16, 700, 50) mm, rotated rx 180 ry 0 rz 90 deg; joints [-18.452, -68.022, 114.764, 155.384, 49.455, -163.415]
  MoveL 218 to (-162.16, 700, -0.5) mm, rotated rx 180 ry 0 rz 90 deg; joints [-18.452, -65.863, 115.091, 156.222, 51.722, -164.734]
  MoveL 219 to (-162.16, 700, 50) mm, rotated rx 180 ry 0 rz 90 deg; joints [-18.452, -68.022, 114.764, 155.384, 49.455, -163.415]
  MoveL 220 to (-162.16, 750, 50) mm, rotated rx -180 ry 0 rz 90 deg; joints [-19.047, -69.77, 117.434, 154.965, 50.461, -163.442]
  MoveL 221 to (-162.16, 750, -0.5) mm, rotated rx 180 ry 0 rz 90 deg; joints [-19.047, -67.525, 117.769, 155.816, 52.807, -164.812]
  MoveL 222 to (-162.16, 750, 50) mm, rotated rx -180 ry 0 rz 90 deg; joints [-19.047, -69.77, 117.434, 154.965, 50.461, -163.442]
  MoveL 223 to (-162.16, 800, 50) mm, rotated rx -180 ry 0 rz 90 deg; joints [-19.679, -71.525, 120.057, 154.485, 51.426, -163.427]
  MoveL 224 to (-162.16, 800, -0.5) mm, rotated rx -180 ry 0 rz 90 deg; joints [-19.679, -69.188, 120.401, 155.353, 53.855, -164.857]
  MoveL 225 to (-162.16, 800, 50) mm, rotated rx -180 ry 0 rz 90 deg; joints [-19.679, -71.525, 120.057, 154.485, 51.426, -163.427]
  MoveL 226 to (-162.16, 850, 50) mm, rotated rx -180 ry 0 rz 90 deg; joints [-20.353, -73.292, 122.634, 153.941, 52.348, -163.368]
  MoveL 227 to (-162.16, 850, -0.5) mm, rotated rx 180 ry 0 rz 90 deg; joints [-20.353, -70.855, 122.989, 154.831, 54.865, -164.867]
  MoveL 228 to (-162.16, 850, 50) mm, rotated rx -180 ry 0 rz 90 deg; joints [-20.353, -73.292, 122.634, 153.941, 52.348, -163.368]
  MoveL 229 to (-162.16, 900, 50) mm, rotated rx 180 ry 0 rz 90 deg; joints [-21.073, -75.075, 125.168, 153.328, 53.227, -163.263]
  MoveL 230 to (-162.16, 900, -0.5) mm, rotated rx -180 ry 0 rz 90 deg; joints [-21.073, -72.532, 125.534, 154.244, 55.838, -164.841]
  MoveL 231 to (-162.16, 900, 50) mm, rotated rx 180 ry 0 rz 90 deg; joints [-21.073, -75.075, 125.168, 153.328, 53.227, -163.263]
  MoveL 232 to (-162.16, 950, 50) mm, rotated rx -180 ry 0 rz 90 deg; joints [-21.843, -76.88, 127.659, 152.643, 54.061, -163.108]
  MoveL 233 to (-162.16, 950, -0.5) mm, rotated rx 180 ry 0 rz 90 deg; joints [-21.843, -74.221, 128.038, 153.59, 56.771, -164.776]
  MoveL 234 to (-162.16, 950, 50) mm, rotated rx -180 ry 0 rz 90 deg; joints [-21.843, -76.88, 127.659, 152.643, 54.061, -163.108]
  MoveL 235 to (-162.16, 1000, 50) mm, rotated rx 180 ry 0 rz 90 deg; joints [-22.668, -78.712, 130.108, 151.878, 54.849, -162.897]
  MoveL 236 to (-162.16, 1000, -0.5) mm, rotated rx 180 ry 0 rz 90 deg; joints [-22.668, -75.929, 130.502, 152.863, 57.664, -164.669]
  MoveL 237 to (-162.16, 1000, 50) mm, rotated rx 180 ry 0 rz 90 deg; joints [-22.668, -78.712, 130.108, 151.878, 54.849, -162.897]
  MoveL 238 to (-162.16, 1050, 50) mm, rotated rx -180 ry 0 rz 90 deg; joints [-23.554, -80.578, 132.516, 151.027, 55.587, -162.624]
  MoveL 239 to (-162.16, 1050, -0.5) mm, rotated rx -180 ry 0 rz 90 deg; joints [-23.554, -77.66, 132.926, 152.056, 58.514, -164.514]
  MoveL 240 to (-162.16, 1050, 50) mm, rotated rx -180 ry 0 rz 90 deg; joints [-23.554, -80.578, 132.516, 151.027, 55.587, -162.624]
  MoveL 241 to (-162.16, 1100, 50) mm, rotated rx 180 ry 0 rz 90 deg; joints [-24.508, -82.486, 134.883, 150.082, 56.275, -162.282]
  MoveL 242 to (-162.16, 1100, -0.5) mm, rotated rx 180 ry 0 rz 90 deg; joints [-24.508, -79.42, 135.311, 151.162, 59.319, -164.307]
  MoveL 243 to (-162.16, 1100, 50) mm, rotated rx 180 ry 0 rz 90 deg; joints [-24.508, -82.486, 134.883, 150.082, 56.275, -162.282]
  MoveL 244 to (-162.16, 1150, 50) mm, rotated rx 180 ry 0 rz 90 deg; joints [-25.537, -84.443, 137.208, 149.032, 56.909, -161.859]
  MoveL 245 to (-162.16, 1150, -0.5) mm, rotated rx -180 ry 0 rz 90 deg; joints [-25.537, -81.218, 137.656, 150.172, 60.078, -164.039]
  MoveL 246 to (-162.16, 1150, 50) mm, rotated rx 180 ry 0 rz 90 deg; joints [-25.537, -84.443, 137.208, 149.032, 56.909, -161.859]
  MoveL 247 to (-162.16, 1200, 50) mm, rotated rx 180 ry 0 rz 90 deg; joints [-26.65, -86.46, 139.491, 147.866, 57.487, -161.344]
  MoveL 248 to (-162.16, 1200, -0.5) mm, rotated rx -180 ry 0 rz 90 deg; joints [-26.65, -83.059, 139.961, 149.076, 60.787, -163.702]
  MoveL 249 to (-162.16, 1200, 50) mm, rotated rx 180 ry 0 rz 90 deg; joints [-26.65, -86.46, 139.491, 147.866, 57.487, -161.344]
  MoveL 250 to (-162.16, 1250, 50) mm, rotated rx -180 ry 0 rz 90 deg; joints [-27.856, -88.547, 141.729, 146.569, 58.006, -160.722]
  MoveL 251 to (-162.16, 1250, -0.5) mm, rotated rx -180 ry 0 rz 90 deg; joints [-27.856, -84.954, 142.225, 147.861, 61.443, -163.284]
  MoveL 252 to (-162.16, 1250, 50) mm, rotated rx -180 ry 0 rz 90 deg; joints [-27.856, -88.547, 141.729, 146.569, 58.006, -160.722]
  MoveL 253 to (-162.16, 1300, 50) mm, rotated rx 180 ry 0 rz 90 deg; joints [-29.167, -90.716, 143.922, 145.125, 58.466, -159.973]
  MoveL 254 to (-162.16, 1300, -0.5) mm, rotated rx -180 ry 0 rz 90 deg; joints [-29.167, -86.914, 144.445, 146.514, 62.045, -162.771]
  MoveL 255 to (-162.16, 1300, 50) mm, rotated rx 180 ry 0 rz 90 deg; joints [-29.167, -90.716, 143.922, 145.125, 58.466, -159.973]
  MoveL 256 to (-162.16, 1350, 50) mm, rotated rx 180 ry 0 rz 90 deg; joints [-30.594, -92.982, 146.066, 143.516, 58.866, -159.075]
  MoveL 257 to (-162.16, 1350, -0.5) mm, rotated rx -180 ry 0 rz 90 deg; joints [-30.594, -88.951, 146.621, 145.018, 62.591, -162.145]
  MoveL 258 to (-162.16, 1350, 50) mm, rotated rx 180 ry 0 rz 90 deg; joints [-30.594, -92.982, 146.066, 143.516, 58.866, -159.075]
  MoveL 259 to (-162.16, 1400, 50) mm, rotated rx 180 ry 0 rz 90 deg; joints [-32.153, -95.362, 148.157, 141.719, 59.208, -158.001]
  MoveL 260 to (-162.16, 1400, -0.5) mm, rotated rx 180 ry 0 rz 90 deg; joints [-32.153, -91.079, 148.748, 143.354, 63.078, -161.385]
  MoveL 261 to (-162.16, 1400, 50) mm, rotated rx 180 ry 0 rz 90 deg; joints [-32.153, -95.362, 148.157, 141.719, 59.208, -158.001]
  MoveL 262 to (-237.84, 50, 50) mm, rotated rx 180 ry 0 rz 90 deg; joints [-11.149, -44.582, 74.995, 158.728, 32.207, -161.767]
  MoveL 263 to (-237.84, 50, -0.5) mm, rotated rx -180 ry 0 rz 90 deg; joints [-11.149, -43.168, 75.294, 159.665, 33.809, -162.884]
  MoveL 264 to (-237.84, 50, 50) mm, rotated rx 180 ry 0 rz 90 deg; joints [-11.149, -44.582, 74.995, 158.728, 32.207, -161.767]
  MoveL 265 to (-237.84, 100, 50) mm, rotated rx 180 ry 0 rz 90 deg; joints [-11.409, -46.666, 78.747, 159.196, 33.844, -162.486]
  MoveL 266 to (-237.84, 100, -0.5) mm, rotated rx -180 ry 0 rz 90 deg; joints [-11.409, -45.208, 79.042, 160.078, 35.488, -163.559]
  MoveL 267 to (-237.84, 100, 50) mm, rotated rx 180 ry 0 rz 90 deg; joints [-11.409, -46.666, 78.747, 159.196, 33.844, -162.486]
  MoveL 268 to (-237.84, 150, 50) mm, rotated rx -180 ry 0 rz 90 deg; joints [-11.681, -48.687, 82.355, 159.549, 35.41, -163.094]
  MoveL 269 to (-237.84, 150, -0.5) mm, rotated rx 180 ry 0 rz 90 deg; joints [-11.681, -47.183, 82.648, 160.388, 37.099, -164.135]
  MoveL 270 to (-237.84, 150, 50) mm, rotated rx -180 ry 0 rz 90 deg; joints [-11.681, -48.687, 82.355, 159.549, 35.41, -163.094]
  MoveL 271 to (-237.84, 200, 50) mm, rotated rx 180 ry 0 rz 90 deg; joints [-11.966, -50.655, 85.838, 159.806, 36.912, -163.612]
  MoveL 272 to (-237.84, 200, -0.5) mm, rotated rx 180 ry 0 rz 90 deg; joints [-11.966, -49.103, 86.13, 160.612, 38.647, -164.631]
  MoveL 273 to (-237.84, 200, 50) mm, rotated rx 180 ry 0 rz 90 deg; joints [-11.966, -50.655, 85.838, 159.806, 36.912, -163.612]
  MoveL 274 to (-237.84, 250, 50) mm, rotated rx 180 ry 0 rz 90 deg; joints [-12.264, -52.578, 89.21, 159.982, 38.356, -164.056]
  MoveL 275 to (-237.84, 250, -0.5) mm, rotated rx 180 ry 0 rz 90 deg; joints [-12.264, -50.976, 89.501, 160.761, 40.14, -165.061]
  MoveL 276 to (-237.84, 250, 50) mm, rotated rx 180 ry 0 rz 90 deg; joints [-12.264, -52.578, 89.21, 159.982, 38.356, -164.056]
  MoveL 277 to (-237.84, 300, 50) mm, rotated rx -180 ry 0 rz 90 deg; joints [-12.578, -54.463, 92.482, 160.086, 39.745, -164.435]
  MoveL 278 to (-237.84, 300, -0.5) mm, rotated rx 180 ry 0 rz 90 deg; joints [-12.578, -52.809, 92.775, 160.844, 41.58, -165.434]
  MoveL 279 to (-237.84, 300, 50) mm, rotated rx -180 ry 0 rz 90 deg; joints [-12.578, -54.463, 92.482, 160.086, 39.745, -164.435]
  MoveL 280 to (-237.84, 350, 50) mm, rotated rx 180 ry 0 rz 90 deg; joints [-12.908, -56.317, 95.665, 160.126, 41.082, -164.759]
  MoveL 281 to (-237.84, 350, -0.5) mm, rotated rx 180 ry 0 rz 90 deg; joints [-12.908, -54.608, 95.96, 160.869, 42.971, -165.758]
  MoveL 282 to (-237.84, 350, 50) mm, rotated rx 180 ry 0 rz 90 deg; joints [-12.908, -56.317, 95.665, 160.126, 41.082, -164.759]
  MoveL 283 to (-237.84, 400, 50) mm, rotated rx 180 ry 0 rz 90 deg; joints [-13.256, -58.146, 98.768, 160.108, 42.371, -165.033]
  MoveL 284 to (-237.84, 400, -0.5) mm, rotated rx 180 ry 0 rz 90 deg; joints [-13.256, -56.378, 99.065, 160.839, 44.317, -166.039]
  MoveL 285 to (-237.84, 400, 50) mm, rotated rx 180 ry 0 rz 90 deg; joints [-13.256, -58.146, 98.768, 160.108, 42.371, -165.033]
  MoveL 286 to (-237.84, 450, 50) mm, rotated rx -180 ry 0 rz 90 deg; joints [-13.623, -59.953, 101.797, 160.035, 43.613, -165.264]
  MoveL 287 to (-237.84, 450, -0.5) mm, rotated rx 180 ry 0 rz 90 deg; joints [-13.623, -58.125, 102.097, 160.759, 45.619, -166.281]
  MoveL 288 to (-237.84, 450, 50) mm, rotated rx -180 ry 0 rz 90 deg; joints [-13.623, -59.953, 101.797, 160.035, 43.613, -165.264]
  MoveL 289 to (-237.84, 500, 50) mm, rotated rx -180 ry 0 rz 90 deg; joints [-14.009, -61.745, 104.758, 159.91, 44.81, -165.454]
  MoveL 290 to (-237.84, 500, -0.5) mm, rotated rx 180 ry 0 rz 90 deg; joints [-14.009, -59.852, 105.063, 160.631, 46.879, -166.488]
  MoveL 291 to (-237.84, 500, 50) mm, rotated rx -180 ry 0 rz 90 deg; joints [-14.009, -61.745, 104.758, 159.91, 44.81, -165.454]
  MoveL 292 to (-237.84, 550, 50) mm, rotated rx 180 ry 0 rz 90 deg; joints [-14.419, -63.526, 107.658, 159.734, 45.962, -165.605]
  MoveL 293 to (-237.84, 550, -0.5) mm, rotated rx -180 ry 0 rz 90 deg; joints [-14.419, -61.563, 107.968, 160.455, 48.099, -166.662]
  MoveL 294 to (-237.84, 550, 50) mm, rotated rx 180 ry 0 rz 90 deg; joints [-14.419, -63.526, 107.658, 159.734, 45.962, -165.605]
  MoveL 295 to (-237.84, 600, 50) mm, rotated rx -180 ry 0 rz 90 deg; joints [-14.852, -65.299, 110.5, 159.509, 47.071, -165.72]
  MoveL 296 to (-237.84, 600, -0.5) mm, rotated rx -180 ry 0 rz 90 deg; joints [-14.852, -63.263, 110.816, 160.233, 49.28, -166.806]
  MoveL 297 to (-237.84, 600, 50) mm, rotated rx -180 ry 0 rz 90 deg; joints [-14.852, -65.299, 110.5, 159.509, 47.071, -165.72]
  MoveL 298 to (-237.84, 650, 50) mm, rotated rx -180 ry 0 rz 90 deg; joints [-15.311, -67.071, 113.288, 159.233, 48.136, -165.798]
  MoveL 299 to (-237.84, 650, -0.5) mm, rotated rx -180 ry 0 rz 90 deg; joints [-15.311, -64.956, 113.611, 159.965, 50.421, -166.92]
  MoveL 300 to (-237.84, 650, 50) mm, rotated rx -180 ry 0 rz 90 deg; joints [-15.311, -67.071, 113.288, 159.233, 48.136, -165.798]
  MoveL 301 to (-237.84, 700, 50) mm, rotated rx 180 ry 0 rz 90 deg; joints [-15.799, -68.844, 116.026, 158.906, 49.157, -165.841]
  MoveL 302 to (-237.84, 700, -0.5) mm, rotated rx -180 ry 0 rz 90 deg; joints [-15.799, -66.645, 116.357, 159.649, 51.523, -167.004]
  MoveL 303 to (-237.84, 700, 50) mm, rotated rx 180 ry 0 rz 90 deg; joints [-15.799, -68.844, 116.026, 158.906, 49.157, -165.841]
  MoveL 304 to (-237.84, 750, 50) mm, rotated rx 180 ry 0 rz 90 deg; joints [-16.318, -70.624, 118.717, 158.527, 50.132, -165.848]
  MoveL 305 to (-237.84, 750, -0.5) mm, rotated rx 180 ry 0 rz 90 deg; joints [-16.318, -68.335, 119.057, 159.283, 52.585, -167.059]
  MoveL 306 to (-237.84, 750, 50) mm, rotated rx 180 ry 0 rz 90 deg; joints [-16.318, -70.624, 118.717, 158.527, 50.132, -165.848]
  MoveL 307 to (-237.84, 800, 50) mm, rotated rx -180 ry 0 rz 90 deg; joints [-16.871, -72.415, 121.363, 158.092, 51.062, -165.816]
  MoveL 308 to (-237.84, 800, -0.5) mm, rotated rx -180 ry 0 rz 90 deg; joints [-16.871, -70.029, 121.713, 158.867, 53.608, -167.083]
  MoveL 309 to (-237.84, 800, 50) mm, rotated rx -180 ry 0 rz 90 deg; joints [-16.871, -72.415, 121.363, 158.092, 51.062, -165.816]
  MoveL 310 to (-237.84, 850, 50) mm, rotated rx 180 ry 0 rz 90 deg; joints [-17.462, -74.224, 123.967, 157.598, 51.944, -165.743]
  MoveL 311 to (-237.84, 850, -0.5) mm, rotated rx 180 ry 0 rz 90 deg; joints [-17.462, -71.732, 124.328, 158.396, 54.588, -167.076]
  MoveL 312 to (-237.84, 850, 50) mm, rotated rx 180 ry 0 rz 90 deg; joints [-17.462, -74.224, 123.967, 157.598, 51.944, -165.743]
  MoveL 313 to (-237.84, 900, 50) mm, rotated rx -180 ry 0 rz 90 deg; joints [-18.095, -76.055, 126.529, 157.042, 52.775, -165.627]
  MoveL 314 to (-237.84, 900, -0.5) mm, rotated rx -180 ry 0 rz 90 deg; joints [-18.095, -73.45, 126.903, 157.867, 55.526, -167.035]
  MoveL 315 to (-237.84, 900, 50) mm, rotated rx -180 ry 0 rz 90 deg; joints [-18.095, -76.055, 126.529, 157.042, 52.775, -165.627]
  MoveL 316 to (-237.84, 950, 50) mm, rotated rx -180 ry 0 rz 90 deg; joints [-18.773, -77.915, 129.053, 156.418, 53.554, -165.462]
  MoveL 317 to (-237.84, 950, -0.5) mm, rotated rx -180 ry 0 rz 90 deg; joints [-18.773, -75.187, 129.44, 157.276, 56.418, -166.957]
  MoveL 318 to (-237.84, 950, 50) mm, rotated rx -180 ry 0 rz 90 deg; joints [-18.773, -77.915, 129.053, 156.418, 53.554, -165.462]
  MoveL 319 to (-237.84, 1000, 50) mm, rotated rx 180 ry 0 rz 90 deg; joints [-19.502, -79.811, 131.537, 155.719, 54.276, -165.243]
  MoveL 320 to (-237.84, 1000, -0.5) mm, rotated rx 180 ry 0 rz 90 deg; joints [-19.502, -76.949, 131.94, 156.616, 57.263, -166.839]
  MoveL 321 to (-237.84, 1000, 50) mm, rotated rx 180 ry 0 rz 90 deg; joints [-19.502, -79.811, 131.537, 155.719, 54.276, -165.243]
  MoveL 322 to (-237.84, 1050, 50) mm, rotated rx 180 ry 0 rz 90 deg; joints [-20.288, -81.752, 133.984, 154.937, 54.937, -164.963]
  MoveL 323 to (-237.84, 1050, -0.5) mm, rotated rx -180 ry 0 rz 90 deg; joints [-20.288, -78.744, 134.405, 155.882, 58.055, -166.674]
  MoveL 324 to (-237.84, 1050, 50) mm, rotated rx 180 ry 0 rz 90 deg; joints [-20.288, -81.752, 133.984, 154.937, 54.937, -164.963]
  MoveL 325 to (-237.84, 1100, 50) mm, rotated rx -180 ry 0 rz 90 deg; joints [-21.136, -83.747, 136.392, 154.064, 55.534, -164.611]
  MoveL 326 to (-237.84, 1100, -0.5) mm, rotated rx 180 ry 0 rz 90 deg; joints [-21.136, -80.579, 136.833, 155.065, 58.793, -166.456]
  MoveL 327 to (-237.84, 1100, 50) mm, rotated rx -180 ry 0 rz 90 deg; joints [-21.136, -83.747, 136.392, 154.064, 55.534, -164.611]
  MoveL 328 to (-237.84, 1150, 50) mm, rotated rx 180 ry 0 rz 90 deg; joints [-22.055, -85.806, 138.763, 153.088, 56.06, -164.177]
  MoveL 329 to (-237.84, 1150, -0.5) mm, rotated rx 180 ry 0 rz 90 deg; joints [-22.055, -82.463, 139.226, 154.155, 59.47, -166.176]
  MoveL 330 to (-237.84, 1150, 50) mm, rotated rx 180 ry 0 rz 90 deg; joints [-22.055, -85.806, 138.763, 153.088, 56.06, -164.177]
  MoveL 331 to (-237.84, 1200, 50) mm, rotated rx 180 ry 0 rz 90 deg; joints [-23.053, -87.944, 141.095, 151.996, 56.509, -163.645]
  MoveL 332 to (-237.84, 1200, -0.5) mm, rotated rx 180 ry 0 rz 90 deg; joints [-23.053, -84.408, 141.583, 153.141, 60.081, -165.824]
  MoveL 333 to (-237.84, 1200, 50) mm, rotated rx 180 ry 0 rz 90 deg; joints [-23.053, -87.944, 141.095, 151.996, 56.509, -163.645]
  MoveL 334 to (-237.84, 1250, 50) mm, rotated rx 180 ry 0 rz 90 deg; joints [-24.14, -90.174, 143.388, 150.769, 56.875, -162.997]
  MoveL 335 to (-237.84, 1250, -0.5) mm, rotated rx 180 ry 0 rz 90 deg; joints [-24.14, -86.426, 143.904, 152.009, 60.619, -165.385]
  MoveL 336 to (-237.84, 1250, 50) mm, rotated rx 180 ry 0 rz 90 deg; joints [-24.14, -90.174, 143.388, 150.769, 56.875, -162.997]
  MoveL 337 to (-237.84, 1300, 50) mm, rotated rx 180 ry 0 rz 90 deg; joints [-25.327, -92.517, 145.638, 149.389, 57.15, -162.206]
  MoveL 338 to (-237.84, 1300, -0.5) mm, rotated rx -180 ry 0 rz 90 deg; joints [-25.327, -88.533, 146.186, 150.742, 61.078, -164.841]
  MoveL 339 to (-237.84, 1300, 50) mm, rotated rx 180 ry 0 rz 90 deg; joints [-25.327, -92.517, 145.638, 149.389, 57.15, -162.206]
  MoveL 340 to (-237.84, 1350, 50) mm, rotated rx 180 ry 0 rz 90 deg; joints [-26.628, -94.993, 147.844, 147.829, 57.327, -161.244]
  MoveL 341 to (-237.84, 1350, -0.5) mm, rotated rx 180 ry 0 rz 90 deg; joints [-26.628, -90.749, 148.429, 149.319, 61.448, -164.168]
  MoveL 342 to (-237.84, 1350, 50) mm, rotated rx 180 ry 0 rz 90 deg; joints [-26.628, -94.993, 147.844, 147.829, 57.327, -161.244]
  MoveL 343 to (-313.52, 50, 50) mm, rotated rx 180 ry 0 rz 90 deg; joints [-9.188, -45.157, 76.033, 162.505, 32.084, -165.047]
  MoveL 344 to (-313.52, 50, -0.5) mm, rotated rx -180 ry 0 rz 90 deg; joints [-9.188, -43.731, 76.331, 163.289, 33.732, -165.981]
  MoveL 345 to (-313.52, 50, 50) mm, rotated rx 180 ry 0 rz 90 deg; joints [-9.188, -45.157, 76.033, 162.505, 32.084, -165.047]
  MoveL 346 to (-313.52, 100, 50) mm, rotated rx 180 ry 0 rz 90 deg; joints [-9.404, -47.236, 79.767, 162.882, 33.719, -165.631]
  MoveL 347 to (-313.52, 100, -0.5) mm, rotated rx 180 ry 0 rz 90 deg; joints [-9.404, -45.765, 80.062, 163.621, 35.41, -166.528]
  MoveL 348 to (-313.52, 100, 50) mm, rotated rx 180 ry 0 rz 90 deg; joints [-9.404, -47.236, 79.767, 162.882, 33.719, -165.631]
  MoveL 349 to (-313.52, 150, 50) mm, rotated rx -180 ry 0 rz 90 deg; joints [-9.63, -49.255, 83.363, 163.165, 35.283, -166.126]
  MoveL 350 to (-313.52, 150, -0.5) mm, rotated rx 180 ry 0 rz 90 deg; joints [-9.63, -47.737, 83.656, 163.868, 37.019, -166.996]
  MoveL 351 to (-313.52, 150, 50) mm, rotated rx -180 ry 0 rz 90 deg; joints [-9.63, -49.255, 83.363, 163.165, 35.283, -166.126]
  MoveL 352 to (-313.52, 200, 50) mm, rotated rx 180 ry 0 rz 90 deg; joints [-9.867, -51.223, 86.837, 163.37, 36.781, -166.546]
  MoveL 353 to (-313.52, 200, -0.5) mm, rotated rx -180 ry 0 rz 90 deg; joints [-9.867, -49.656, 87.129, 164.045, 38.565, -167.399]
  MoveL 354 to (-313.52, 200, 50) mm, rotated rx 180 ry 0 rz 90 deg; joints [-9.867, -51.223, 86.837, 163.37, 36.781, -166.546]
  MoveL 355 to (-313.52, 250, 50) mm, rotated rx 180 ry 0 rz 90 deg; joints [-10.116, -53.148, 90.204, 163.507, 38.219, -166.905]
  MoveL 356 to (-313.52, 250, -0.5) mm, rotated rx -180 ry 0 rz 90 deg; joints [-10.116, -51.531, 90.495, 164.16, 40.053, -167.747]
  MoveL 357 to (-313.52, 250, 50) mm, rotated rx 180 ry 0 rz 90 deg; joints [-10.116, -53.148, 90.204, 163.507, 38.219, -166.905]
  MoveL 358 to (-313.52, 300, 50) mm, rotated rx -180 ry 0 rz 90 deg; joints [-10.378, -55.039, 93.474, 163.585, 39.601, -167.211]
  MoveL 359 to (-313.52, 300, -0.5) mm, rotated rx -180 ry 0 rz 90 deg; joints [-10.378, -53.368, 93.767, 164.222, 41.488, -168.049]
  MoveL 360 to (-313.52, 300, 50) mm, rotated rx -180 ry 0 rz 90 deg; joints [-10.378, -55.039, 93.474, 163.585, 39.601, -167.211]
  MoveL 361 to (-313.52, 350, 50) mm, rotated rx 180 ry 0 rz 90 deg; joints [-10.653, -56.9, 96.658, 163.611, 40.931, -167.472]
  MoveL 362 to (-313.52, 350, -0.5) mm, rotated rx 180 ry 0 rz 90 deg; joints [-10.653, -55.172, 96.953, 164.235, 42.874, -168.311]
  MoveL 363 to (-313.52, 350, 50) mm, rotated rx 180 ry 0 rz 90 deg; joints [-10.653, -56.9, 96.658, 163.611, 40.931, -167.472]
  MoveL 364 to (-313.52, 400, 50) mm, rotated rx -180 ry 0 rz 90 deg; joints [-10.943, -58.737, 99.763, 163.587, 42.21, -167.692]
  MoveL 365 to (-313.52, 400, -0.5) mm, rotated rx 180 ry 0 rz 90 deg; joints [-10.943, -56.95, 100.061, 164.203, 44.213, -168.537]
  MoveL 366 to (-313.52, 400, 50) mm, rotated rx -180 ry 0 rz 90 deg; joints [-10.943, -58.737, 99.763, 163.587, 42.21, -167.692]
  MoveL 367 to (-313.52, 450, 50) mm, rotated rx -180 ry 0 rz 90 deg; joints [-11.249, -60.556, 102.798, 163.518, 43.44, -167.876]
  MoveL 368 to (-313.52, 450, -0.5) mm, rotated rx -180 ry 0 rz 90 deg; joints [-11.249, -58.706, 103.1, 164.129, 45.507, -168.731]
  MoveL 369 to (-313.52, 450, 50) mm, rotated rx -180 ry 0 rz 90 deg; joints [-11.249, -60.556, 102.798, 163.518, 43.44, -167.876]
  MoveL 370 to (-313.52, 500, 50) mm, rotated rx -180 ry 0 rz 90 deg; joints [-11.573, -62.362, 105.767, 163.406, 44.623, -168.025]
  MoveL 371 to (-313.52, 500, -0.5) mm, rotated rx 180 ry 0 rz 90 deg; joints [-11.573, -60.445, 106.073, 164.015, 46.758, -168.896]
  MoveL 372 to (-313.52, 500, 50) mm, rotated rx -180 ry 0 rz 90 deg; joints [-11.573, -62.362, 105.767, 163.406, 44.623, -168.025]
  MoveL 373 to (-313.52, 550, 50) mm, rotated rx 180 ry 0 rz 90 deg; joints [-11.915, -64.158, 108.676, 163.251, 45.76, -168.142]
  MoveL 374 to (-313.52, 550, -0.5) mm, rotated rx 180 ry 0 rz 90 deg; joints [-11.915, -62.17, 108.988, 163.861, 47.966, -169.034]
  MoveL 375 to (-313.52, 550, 50) mm, rotated rx 180 ry 0 rz 90 deg; joints [-11.915, -64.158, 108.676, 163.251, 45.76, -168.142]
  MoveL 376 to (-313.52, 600, 50) mm, rotated rx 180 ry 0 rz 90 deg; joints [-12.278, -65.95, 111.53, 163.053, 46.851, -168.228]
  MoveL 377 to (-313.52, 600, -0.5) mm, rotated rx -180 ry 0 rz 90 deg; joints [-12.278, -63.886, 111.849, 163.668, 49.134, -169.146]
  MoveL 378 to (-313.52, 600, 50) mm, rotated rx 180 ry 0 rz 90 deg; joints [-12.278, -65.95, 111.53, 163.053, 46.851, -168.228]
  MoveL 379 to (-313.52, 650, 50) mm, rotated rx -180 ry 0 rz 90 deg; joints [-12.664, -67.743, 114.333, 162.813, 47.894, -168.284]
  MoveL 380 to (-313.52, 650, -0.5) mm, rotated rx 180 ry 0 rz 90 deg; joints [-12.664, -65.597, 114.659, 163.435, 50.26, -169.233]
  MoveL 381 to (-313.52, 650, 50) mm, rotated rx -180 ry 0 rz 90 deg; joints [-12.664, -67.743, 114.333, 162.813, 47.894, -168.284]
  MoveL 382 to (-313.52, 700, 50) mm, rotated rx 180 ry 0 rz 90 deg; joints [-13.074, -69.541, 117.088, 162.529, 48.891, -168.308]
  MoveL 383 to (-313.52, 700, -0.5) mm, rotated rx 180 ry 0 rz 90 deg; joints [-13.074, -67.308, 117.422, 163.162, 51.344, -169.295]
  MoveL 384 to (-313.52, 700, 50) mm, rotated rx 180 ry 0 rz 90 deg; joints [-13.074, -69.541, 117.088, 162.529, 48.891, -168.308]
  MoveL 385 to (-313.52, 750, 50) mm, rotated rx -180 ry 0 rz 90 deg; joints [-13.511, -71.35, 119.797, 162.199, 49.838, -168.301]
  MoveL 386 to (-313.52, 750, -0.5) mm, rotated rx -180 ry 0 rz 90 deg; joints [-13.511, -69.022, 120.141, 162.847, 52.386, -169.331]
  MoveL 387 to (-313.52, 750, 50) mm, rotated rx -180 ry 0 rz 90 deg; joints [-13.511, -71.35, 119.797, 162.199, 49.838, -168.301]
  MoveL 388 to (-313.52, 800, 50) mm, rotated rx 180 ry 0 rz 90 deg; joints [-13.977, -73.174, 122.465, 161.822, 50.734, -168.259]
  MoveL 389 to (-313.52, 800, -0.5) mm, rotated rx -180 ry 0 rz 90 deg; joints [-13.977, -70.745, 122.819, 162.487, 53.384, -169.341]
  MoveL 390 to (-313.52, 800, 50) mm, rotated rx 180 ry 0 rz 90 deg; joints [-13.977, -73.174, 122.465, 161.822, 50.734, -168.259]
  MoveL 391 to (-313.52, 850, 50) mm, rotated rx 180 ry 0 rz 90 deg; joints [-14.477, -75.021, 125.092, 161.392, 51.577, -168.182]
  MoveL 392 to (-313.52, 850, -0.5) mm, rotated rx 180 ry 0 rz 90 deg; joints [-14.477, -72.481, 125.458, 162.08, 54.337, -169.323]
  MoveL 393 to (-313.52, 850, 50) mm, rotated rx 180 ry 0 rz 90 deg; joints [-14.477, -75.021, 125.092, 161.392, 51.577, -168.182]
  MoveL 394 to (-313.52, 900, 50) mm, rotated rx 180 ry 0 rz 90 deg; joints [-15.012, -76.896, 127.68, 160.908, 52.363, -168.065]
  MoveL 395 to (-313.52, 900, -0.5) mm, rotated rx -180 ry 0 rz 90 deg; joints [-15.012, -74.236, 128.06, 161.622, 55.241, -169.275]
  MoveL 396 to (-313.52, 900, 50) mm, rotated rx 180 ry 0 rz 90 deg; joints [-15.012, -76.896, 127.68, 160.908, 52.363, -168.065]
  MoveL 397 to (-313.52, 950, 50) mm, rotated rx -180 ry 0 rz 90 deg; joints [-15.587, -78.807, 130.232, 160.362, 53.087, -167.904]
  MoveL 398 to (-313.52, 950, -0.5) mm, rotated rx -180 ry 0 rz 90 deg; joints [-15.587, -76.017, 130.627, 161.109, 56.094, -169.193]
  MoveL 399 to (-313.52, 950, 50) mm, rotated rx -180 ry 0 rz 90 deg; joints [-15.587, -78.807, 130.232, 160.362, 53.087, -167.904]
  MoveL 400 to (-313.52, 1000, 50) mm, rotated rx 180 ry 0 rz 90 deg; joints [-16.208, -80.762, 132.748, 159.749, 53.745, -167.692]
  MoveL 401 to (-313.52, 1000, -0.5) mm, rotated rx 180 ry 0 rz 90 deg; joints [-16.208, -77.83, 133.16, 160.535, 56.891, -169.073]
  MoveL 402 to (-313.52, 1000, 50) mm, rotated rx 180 ry 0 rz 90 deg; joints [-16.208, -80.762, 132.748, 159.749, 53.745, -167.692]
  MoveL 403 to (-313.52, 1050, 50) mm, rotated rx -180 ry 0 rz 90 deg; joints [-16.878, -82.772, 135.229, 159.061, 54.331, -167.422]
  MoveL 404 to (-313.52, 1050, -0.5) mm, rotated rx -180 ry 0 rz 90 deg; joints [-16.878, -79.684, 135.66, 159.894, 57.627, -168.91]
  MoveL 405 to (-313.52, 1050, 50) mm, rotated rx -180 ry 0 rz 90 deg; joints [-16.878, -82.772, 135.229, 159.061, 54.331, -167.422]
  MoveL 406 to (-313.52, 1100, 50) mm, rotated rx -180 ry 0 rz 90 deg; joints [-17.604, -84.849, 137.676, 158.288, 54.836, -167.084]
  MoveL 407 to (-313.52, 1100, -0.5) mm, rotated rx 180 ry 0 rz 90 deg; joints [-17.604, -81.588, 138.128, 159.177, 58.296, -168.697]
  MoveL 408 to (-313.52, 1100, 50) mm, rotated rx -180 ry 0 rz 90 deg; joints [-17.604, -84.849, 137.676, 158.288, 54.836, -167.084]
  MoveL 409 to (-313.52, 1150, 50) mm, rotated rx 180 ry 0 rz 90 deg; joints [-18.393, -87.005, 140.088, 157.417, 55.251, -166.664]
  MoveL 410 to (-313.52, 1150, -0.5) mm, rotated rx 180 ry 0 rz 90 deg; joints [-18.393, -83.555, 140.565, 158.375, 58.889, -168.424]
  MoveL 411 to (-313.52, 1150, 50) mm, rotated rx 180 ry 0 rz 90 deg; joints [-18.393, -87.005, 140.088, 157.417, 55.251, -166.664]
  MoveL 412 to (-313.52, 1200, 50) mm, rotated rx -180 ry 0 rz 90 deg; joints [-19.253, -89.259, 142.465, 156.435, 55.567, -166.146]
  MoveL 413 to (-313.52, 1200, -0.5) mm, rotated rx -180 ry 0 rz 90 deg; joints [-19.253, -85.599, 142.969, 157.475, 59.399, -168.079]
  MoveL 414 to (-313.52, 1200, 50) mm, rotated rx -180 ry 0 rz 90 deg; joints [-19.253, -89.259, 142.465, 156.435, 55.567, -166.146]
  MoveL 415 to (-313.52, 1250, 50) mm, rotated rx -180 ry 0 rz 90 deg; joints [-20.194, -91.631, 144.806, 155.321, 55.769, -165.507]
  MoveL 416 to (-313.52, 1250, -0.5) mm, rotated rx -180 ry 0 rz 90 deg; joints [-20.194, -87.738, 145.342, 156.462, 59.812, -167.645]
  MoveL 417 to (-313.52, 1250, 50) mm, rotated rx -180 ry 0 rz 90 deg; joints [-20.194, -91.631, 144.806, 155.321, 55.769, -165.507]
  MoveL 418 to (-313.52, 1300, 50) mm, rotated rx -180 ry 0 rz 90 deg; joints [-21.228, -94.146, 147.109, 154.052, 55.843, -164.719]
  MoveL 419 to (-313.52, 1300, -0.5) mm, rotated rx -180 ry 0 rz 90 deg; joints [-21.228, -89.992, 147.681, 155.317, 60.115, -167.102]
  MoveL 420 to (-313.52, 1300, 50) mm, rotated rx -180 ry 0 rz 90 deg; joints [-21.228, -94.146, 147.109, 154.052, 55.843, -164.719]
  MoveL 421 to (-389.2, 50, 50) mm, rotated rx 180 ry 0 rz 90 deg; joints [-7.205, -45.617, 76.862, 166.302, 31.983, -168.319]
  MoveL 422 to (-389.2, 50, -0.5) mm, rotated rx -180 ry 0 rz 90 deg; joints [-7.205, -44.181, 77.159, 166.924, 33.669, -169.06]
  MoveL 423 to (-389.2, 50, 50) mm, rotated rx 180 ry 0 rz 90 deg; joints [-7.205, -45.617, 76.862, 166.302, 31.983, -168.319]
  MoveL 424 to (-389.2, 100, 50) mm, rotated rx 180 ry 0 rz 90 deg; joints [-7.376, -47.693, 80.584, 166.593, 33.617, -168.772]
  MoveL 425 to (-389.2, 100, -0.5) mm, rotated rx 180 ry 0 rz 90 deg; joints [-7.376, -46.211, 80.878, 167.179, 35.346, -169.484]
  MoveL 426 to (-389.2, 100, 50) mm, rotated rx 180 ry 0 rz 90 deg; joints [-7.376, -47.693, 80.584, 166.593, 33.617, -168.772]
  MoveL 427 to (-389.2, 150, 50) mm, rotated rx 180 ry 0 rz 90 deg; joints [-7.554, -49.71, 84.17, 166.81, 35.178, -169.155]
  MoveL 428 to (-389.2, 150, -0.5) mm, rotated rx -180 ry 0 rz 90 deg; joints [-7.554, -48.181, 84.462, 167.368, 36.953, -169.847]
  MoveL 429 to (-389.2, 150, 50) mm, rotated rx 180 ry 0 rz 90 deg; joints [-7.554, -49.71, 84.17, 166.81, 35.178, -169.155]
  MoveL 430 to (-389.2, 200, 50) mm, rotated rx -180 ry 0 rz 90 deg; joints [-7.742, -51.679, 87.638, 166.965, 36.673, -169.481]
  MoveL 431 to (-389.2, 200, -0.5) mm, rotated rx 180 ry 0 rz 90 deg; joints [-7.742, -50.101, 87.93, 167.502, 38.496, -170.158]
  MoveL 432 to (-389.2, 200, 50) mm, rotated rx -180 ry 0 rz 90 deg; joints [-7.742, -51.679, 87.638, 166.965, 36.673, -169.481]
  MoveL 433 to (-389.2, 250, 50) mm, rotated rx -180 ry 0 rz 90 deg; joints [-7.938, -53.608, 91.001, 167.068, 38.106, -169.758]
  MoveL 434 to (-389.2, 250, -0.5) mm, rotated rx 180 ry 0 rz 90 deg; joints [-7.938, -51.977, 91.293, 167.588, 39.982, -170.428]
  MoveL 435 to (-389.2, 250, 50) mm, rotated rx -180 ry 0 rz 90 deg; joints [-7.938, -53.608, 91.001, 167.068, 38.106, -169.758]
  MoveL 436 to (-389.2, 300, 50) mm, rotated rx -180 ry 0 rz 90 deg; joints [-8.145, -55.502, 94.27, 167.125, 39.482, -169.995]
  MoveL 437 to (-389.2, 300, -0.5) mm, rotated rx -180 ry 0 rz 90 deg; joints [-8.145, -53.818, 94.564, 167.632, 41.413, -170.661]
  MoveL 438 to (-389.2, 300, 50) mm, rotated rx -180 ry 0 rz 90 deg; joints [-8.145, -55.502, 94.27, 167.125, 39.482, -169.995]
  MoveL 439 to (-389.2, 350, 50) mm, rotated rx 180 ry 0 rz 90 deg; joints [-8.363, -57.369, 97.455, 167.139, 40.804, -170.195]
  MoveL 440 to (-389.2, 350, -0.5) mm, rotated rx 180 ry 0 rz 90 deg; joints [-8.363, -55.627, 97.751, 167.637, 42.793, -170.863]
  MoveL 441 to (-389.2, 350, 50) mm, rotated rx 180 ry 0 rz 90 deg; joints [-8.363, -57.369, 97.455, 167.139, 40.804, -170.195]
  MoveL 442 to (-389.2, 400, 50) mm, rotated rx 180 ry 0 rz 90 deg; joints [-8.593, -59.215, 100.564, 167.116, 42.075, -170.364]
  MoveL 443 to (-389.2, 400, -0.5) mm, rotated rx 180 ry 0 rz 90 deg; joints [-8.593, -57.412, 100.863, 167.607, 44.126, -171.037]
  MoveL 444 to (-389.2, 400, 50) mm, rotated rx 180 ry 0 rz 90 deg; joints [-8.593, -59.215, 100.564, 167.116, 42.075, -170.364]
  MoveL 445 to (-389.2, 450, 50) mm, rotated rx -180 ry 0 rz 90 deg; joints [-8.836, -61.043, 103.603, 167.056, 43.295, -170.503]
  MoveL 446 to (-389.2, 450, -0.5) mm, rotated rx -180 ry 0 rz 90 deg; joints [-8.836, -59.176, 103.906, 167.544, 45.413, -171.186]
  MoveL 447 to (-389.2, 450, 50) mm, rotated rx -180 ry 0 rz 90 deg; joints [-8.836, -61.043, 103.603, 167.056, 43.295, -170.503]
  MoveL 448 to (-389.2, 500, 50) mm, rotated rx 180 ry 0 rz 90 deg; joints [-9.093, -62.86, 106.579, 166.962, 44.467, -170.616]
  MoveL 449 to (-389.2, 500, -0.5) mm, rotated rx -180 ry 0 rz 90 deg; joints [-9.093, -60.924, 106.887, 167.449, 46.655, -171.312]
  MoveL 450 to (-389.2, 500, 50) mm, rotated rx 180 ry 0 rz 90 deg; joints [-9.093, -62.86, 106.579, 166.962, 44.467, -170.616]
  MoveL 451 to (-389.2, 550, 50) mm, rotated rx -180 ry 0 rz 90 deg; joints [-9.365, -64.67, 109.497, 166.833, 45.59, -170.703]
  MoveL 452 to (-389.2, 550, -0.5) mm, rotated rx 180 ry 0 rz 90 deg; joints [-9.365, -62.661, 109.811, 167.322, 47.855, -171.416]
  MoveL 453 to (-389.2, 550, 50) mm, rotated rx -180 ry 0 rz 90 deg; joints [-9.365, -64.67, 109.497, 166.833, 45.59, -170.703]
  MoveL 454 to (-389.2, 600, 50) mm, rotated rx -180 ry 0 rz 90 deg; joints [-9.654, -66.479, 112.362, 166.67, 46.665, -170.765]
  MoveL 455 to (-389.2, 600, -0.5) mm, rotated rx -180 ry 0 rz 90 deg; joints [-9.654, -64.391, 112.682, 167.164, 49.011, -171.5]
  MoveL 456 to (-389.2, 600, 50) mm, rotated rx -180 ry 0 rz 90 deg; joints [-9.654, -66.479, 112.362, 166.67, 46.665, -170.765]
  MoveL 457 to (-389.2, 650, 50) mm, rotated rx -180 ry 0 rz 90 deg; joints [-9.96, -68.29, 115.177, 166.473, 47.69, -170.802]
  MoveL 458 to (-389.2, 650, -0.5) mm, rotated rx -180 ry 0 rz 90 deg; joints [-9.96, -66.118, 115.505, 166.974, 50.123, -171.563]
  MoveL 459 to (-389.2, 650, 50) mm, rotated rx -180 ry 0 rz 90 deg; joints [-9.96, -68.29, 115.177, 166.473, 47.69, -170.802]
  MoveL 460 to (-389.2, 700, 50) mm, rotated rx 180 ry 0 rz 90 deg; joints [-10.287, -70.109, 117.945, 166.241, 48.665, -170.813]
  MoveL 461 to (-389.2, 700, -0.5) mm, rotated rx 180 ry 0 rz 90 deg; joints [-10.287, -67.847, 118.282, 166.752, 51.192, -171.607]
  MoveL 462 to (-389.2, 700, 50) mm, rotated rx 180 ry 0 rz 90 deg; joints [-10.287, -70.109, 117.945, 166.241, 48.665, -170.813]
  MoveL 463 to (-389.2, 750, 50) mm, rotated rx 180 ry 0 rz 90 deg; joints [-10.636, -71.942, 120.671, 165.971, 49.587, -170.799]
  MoveL 464 to (-389.2, 750, -0.5) mm, rotated rx -180 ry 0 rz 90 deg; joints [-10.636, -69.582, 121.018, 166.495, 52.216, -171.629]
  MoveL 465 to (-389.2, 750, 50) mm, rotated rx 180 ry 0 rz 90 deg; joints [-10.636, -71.942, 120.671, 165.971, 49.587, -170.799]
  MoveL 466 to (-389.2, 800, 50) mm, rotated rx 180 ry 0 rz 90 deg; joints [-11.009, -73.795, 123.356, 165.662, 50.454, -170.756]
  MoveL 467 to (-389.2, 800, -0.5) mm, rotated rx 180 ry 0 rz 90 deg; joints [-11.009, -71.329, 123.714, 166.202, 53.193, -171.63]
  MoveL 468 to (-389.2, 800, 50) mm, rotated rx 180 ry 0 rz 90 deg; joints [-11.009, -73.795, 123.356, 165.662, 50.454, -170.756]
  MoveL 469 to (-389.2, 850, 50) mm, rotated rx -180 ry 0 rz 90 deg; joints [-11.408, -75.674, 126.003, 165.31, 51.262, -170.684]
  MoveL 470 to (-389.2, 850, -0.5) mm, rotated rx 180 ry 0 rz 90 deg; joints [-11.408, -73.093, 126.374, 165.87, 54.12, -171.607]
  MoveL 471 to (-389.2, 850, 50) mm, rotated rx -180 ry 0 rz 90 deg; joints [-11.408, -75.674, 126.003, 165.31, 51.262, -170.684]
  MoveL 472 to (-389.2, 900, 50) mm, rotated rx 180 ry 0 rz 90 deg; joints [-11.838, -77.587, 128.614, 164.912, 52.006, -170.577]
  MoveL 473 to (-389.2, 900, -0.5) mm, rotated rx -180 ry 0 rz 90 deg; joints [-11.838, -74.881, 128.999, 165.496, 54.994, -171.559]
  MoveL 474 to (-389.2, 900, 50) mm, rotated rx 180 ry 0 rz 90 deg; joints [-11.838, -77.587, 128.614, 164.912, 52.006, -170.577]
  MoveL 475 to (-389.2, 950, 50) mm, rotated rx 180 ry 0 rz 90 deg; joints [-12.3, -79.542, 131.19, 164.462, 52.681, -170.432]
  MoveL 476 to (-389.2, 950, -0.5) mm, rotated rx 180 ry 0 rz 90 deg; joints [-12.3, -76.7, 131.591, 165.076, 55.811, -171.482]
  MoveL 477 to (-389.2, 950, 50) mm, rotated rx 180 ry 0 rz 90 deg; joints [-12.3, -79.542, 131.19, 164.462, 52.681, -170.432]
  MoveL 478 to (-389.2, 1000, 50) mm, rotated rx -180 ry 0 rz 90 deg; joints [-12.799, -81.549, 133.733, 163.956, 53.28, -170.244]
  MoveL 479 to (-389.2, 1000, -0.5) mm, rotated rx 180 ry 0 rz 90 deg; joints [-12.799, -78.557, 134.152, 164.605, 56.564, -171.373]
  MoveL 480 to (-389.2, 1000, 50) mm, rotated rx -180 ry 0 rz 90 deg; joints [-12.799, -81.549, 133.733, 163.956, 53.28, -170.244]
  MoveL 481 to (-389.2, 1050, 50) mm, rotated rx 180 ry 0 rz 90 deg; joints [-13.34, -83.621, 136.243, 163.385, 53.795, -170.004]
  MoveL 482 to (-389.2, 1050, -0.5) mm, rotated rx -180 ry 0 rz 90 deg; joints [-13.34, -80.463, 136.683, 164.077, 57.248, -171.226]
  MoveL 483 to (-389.2, 1050, 50) mm, rotated rx 180 ry 0 rz 90 deg; joints [-13.34, -83.621, 136.243, 163.385, 53.795, -170.004]
  MoveL 484 to (-389.2, 1100, 50) mm, rotated rx -180 ry 0 rz 90 deg; joints [-13.928, -85.77, 138.722, 162.74, 54.214, -169.702]
  MoveL 485 to (-389.2, 1100, -0.5) mm, rotated rx -180 ry 0 rz 90 deg; joints [-13.928, -82.43, 139.185, 163.484, 57.852, -171.034]
  MoveL 486 to (-389.2, 1100, 50) mm, rotated rx -180 ry 0 rz 90 deg; joints [-13.928, -85.77, 138.722, 162.74, 54.214, -169.702]
  MoveL 487 to (-389.2, 1150, 50) mm, rotated rx 180 ry 0 rz 90 deg; joints [-14.568, -88.014, 141.17, 162.009, 54.524, -169.327]
  MoveL 488 to (-389.2, 1150, -0.5) mm, rotated rx 180 ry 0 rz 90 deg; joints [-14.568, -84.471, 141.658, 162.817, 58.367, -170.788]
  MoveL 489 to (-389.2, 1150, 50) mm, rotated rx 180 ry 0 rz 90 deg; joints [-14.568, -88.014, 141.17, 162.009, 54.524, -169.327]
  MoveL 490 to (-389.2, 1200, 50) mm, rotated rx -180 ry 0 rz 90 deg; joints [-15.269, -90.374, 143.585, 161.177, 54.709, -168.859]
  MoveL 491 to (-389.2, 1200, -0.5) mm, rotated rx -180 ry 0 rz 90 deg; joints [-15.269, -86.606, 144.104, 162.064, 58.778, -170.476]
  MoveL 492 to (-389.2, 1200, 50) mm, rotated rx -180 ry 0 rz 90 deg; joints [-15.269, -90.374, 143.585, 161.177, 54.709, -168.859]
  MoveL 493 to (-33.64, 230, 50) mm, rotated rx -180 ry 0 rz 90 deg; joints [-17.705, -49.723, 84.193, 150.574, 38.245, -156.107]
  MoveL 494 to (-33.64, 230, -0.5) mm, rotated rx 180 ry 0 rz 90 deg; joints [-17.705, -48.194, 84.485, 151.659, 39.84, -157.503]
  MoveL 495 to (-33.64, 230, 50) mm, rotated rx -180 ry 0 rz 90 deg; joints [-17.705, -49.723, 84.193, 150.574, 38.245, -156.107]
  MoveL 496 to (-63.64, 230, 50) mm, rotated rx 180 ry 0 rz 90 deg; joints [-16.907, -50.081, 84.826, 151.928, 38.17, -157.252]
  MoveL 497 to (-63.64, 230, -0.5) mm, rotated rx 180 ry 0 rz 90 deg; joints [-16.907, -48.543, 85.118, 152.974, 39.792, -158.597]
  MoveL 498 to (-63.64, 230, 50) mm, rotated rx 180 ry 0 rz 90 deg; joints [-16.907, -50.081, 84.826, 151.928, 38.17, -157.252]
  MoveL 499 to (-109.34, 230, 50) mm, rotated rx 180 ry 0 rz 90 deg; joints [-15.677, -50.592, 85.728, 154.003, 38.06, -158.994]
  MoveL 500 to (-109.34, 230, -0.5) mm, rotated rx 180 ry 0 rz 90 deg; joints [-15.677, -49.042, 86.02, 154.986, 39.723, -160.258]
  MoveL 501 to (-109.34, 230, 50) mm, rotated rx 180 ry 0 rz 90 deg; joints [-15.677, -50.592, 85.728, 154.003, 38.06, -158.994]
  MoveL 502 to (-139.34, 230, 50) mm, rotated rx 180 ry 0 rz 90 deg; joints [-14.862, -50.906, 86.281, 155.374, 37.991, -160.137]
  MoveL 503 to (-139.34, 230, -0.5) mm, rotated rx 180 ry 0 rz 90 deg; joints [-14.862, -49.348, 86.572, 156.314, 39.679, -161.344]
  MoveL 504 to (-139.34, 230, 50) mm, rotated rx 180 ry 0 rz 90 deg; joints [-14.862, -50.906, 86.281, 155.374, 37.991, -160.137]
  MoveL 505 to (-185.04, 230, 50) mm, rotated rx 180 ry 0 rz 90 deg; joints [-13.608, -51.351, 87.062, 157.475, 37.891, -161.877]
  MoveL 506 to (-185.04, 230, -0.5) mm, rotated rx -180 ry 0 rz 90 deg; joints [-13.608, -49.781, 87.353, 158.347, 39.616, -162.995]
  MoveL 507 to (-185.04, 230, 50) mm, rotated rx 180 ry 0 rz 90 deg; joints [-13.608, -51.351, 87.062, 157.475, 37.891, -161.877]
  MoveL 508 to (-215.04, 230, 50) mm, rotated rx 180 ry 0 rz 90 deg; joints [-12.778, -51.62, 87.535, 158.862, 37.83, -163.019]
  MoveL 509 to (-215.04, 230, -0.5) mm, rotated rx -180 ry 0 rz 90 deg; joints [-12.778, -50.043, 87.826, 159.687, 39.577, -164.076]
  MoveL 510 to (-215.04, 230, 50) mm, rotated rx 180 ry 0 rz 90 deg; joints [-12.778, -51.62, 87.535, 158.862, 37.83, -163.019]
  MoveL 511 to (-260.74, 230, 50) mm, rotated rx 180 ry 0 rz 90 deg; joints [-11.502, -51.997, 88.196, 160.988, 37.742, -164.758]
  MoveL 512 to (-260.74, 230, -0.5) mm, rotated rx 180 ry 0 rz 90 deg; joints [-11.502, -50.411, 88.487, 161.739, 39.522, -165.72]
  MoveL 513 to (-260.74, 230, 50) mm, rotated rx 180 ry 0 rz 90 deg; joints [-11.502, -51.997, 88.196, 160.988, 37.742, -164.758]
  MoveL 514 to (-290.74, 230, 50) mm, rotated rx 180 ry 0 rz 90 deg; joints [-10.659, -52.223, 88.59, 162.39, 37.689, -165.9]
  MoveL 515 to (-290.74, 230, -0.5) mm, rotated rx 180 ry 0 rz 90 deg; joints [-10.659, -50.631, 88.882, 163.091, 39.488, -166.797]
  MoveL 516 to (-290.74, 230, 50) mm, rotated rx 180 ry 0 rz 90 deg; joints [-10.659, -52.223, 88.59, 162.39, 37.689, -165.9]
  MoveL 517 to (-336.44, 230, 50) mm, rotated rx -180 ry 0 rz 90 deg; joints [-9.365, -52.533, 89.132, 164.538, 37.615, -167.641]
  MoveL 518 to (-336.44, 230, -0.5) mm, rotated rx 180 ry 0 rz 90 deg; joints [-9.365, -50.932, 89.423, 165.16, 39.441, -168.435]
  MoveL 519 to (-336.44, 230, 50) mm, rotated rx -180 ry 0 rz 90 deg; joints [-9.365, -52.533, 89.132, 164.538, 37.615, -167.641]
  MoveL 520 to (-366.44, 230, 50) mm, rotated rx -180 ry 0 rz 90 deg; joints [-8.51, -52.715, 89.448, 165.955, 37.571, -168.785]
  MoveL 521 to (-366.44, 230, -0.5) mm, rotated rx -180 ry 0 rz 90 deg; joints [-8.51, -51.109, 89.74, 166.522, 39.414, -169.51]
  MoveL 522 to (-366.44, 230, 50) mm, rotated rx -180 ry 0 rz 90 deg; joints [-8.51, -52.715, 89.448, 165.955, 37.571, -168.785]
  MoveL 523 to (-33.64, 420, 50) mm, rotated rx -180 ry 0 rz 90 deg; joints [-19.467, -56.706, 96.328, 151.001, 43.429, -158.073]
  MoveL 524 to (-33.64, 420, -0.5) mm, rotated rx -180 ry 0 rz 90 deg; joints [-19.467, -54.985, 96.623, 151.987, 45.2, -159.451]
  MoveL 525 to (-33.64, 420, 50) mm, rotated rx -180 ry 0 rz 90 deg; joints [-19.467, -56.706, 96.328, 151.001, 43.429, -158.073]
  MoveL 526 to (-63.64, 420, 50) mm, rotated rx -180 ry 0 rz 90 deg; joints [-18.6, -57.074, 96.954, 152.306, 43.339, -159.106]
  MoveL 527 to (-63.64, 420, -0.5) mm, rotated rx -180 ry 0 rz 90 deg; joints [-18.6, -55.342, 97.25, 153.258, 45.143, -160.435]
  MoveL 528 to (-63.64, 420, 50) mm, rotated rx -180 ry 0 rz 90 deg; joints [-18.6, -57.074, 96.954, 152.306, 43.339, -159.106]
  MoveL 529 to (-109.34, 420, 50) mm, rotated rx -180 ry 0 rz 90 deg; joints [-17.263, -57.602, 97.85, 154.313, 43.207, -160.681]
  MoveL 530 to (-109.34, 420, -0.5) mm, rotated rx 180 ry 0 rz 90 deg; joints [-17.263, -55.853, 98.146, 155.212, 45.058, -161.933]
  MoveL 531 to (-109.34, 420, 50) mm, rotated rx -180 ry 0 rz 90 deg; joints [-17.263, -57.602, 97.85, 154.313, 43.207, -160.681]
  MoveL 532 to (-139.34, 420, 50) mm, rotated rx 180 ry 0 rz 90 deg; joints [-16.374, -57.927, 98.399, 155.644, 43.124, -161.716]
  MoveL 533 to (-139.34, 420, -0.5) mm, rotated rx 180 ry 0 rz 90 deg; joints [-16.374, -56.167, 98.695, 156.506, 45.004, -162.916]
  MoveL 534 to (-139.34, 420, 50) mm, rotated rx 180 ry 0 rz 90 deg; joints [-16.374, -57.927, 98.399, 155.644, 43.124, -161.716]
  MoveL 535 to (-185.04, 420, 50) mm, rotated rx -180 ry 0 rz 90 deg; joints [-15.005, -58.388, 99.177, 157.692, 43.003, -163.298]
  MoveL 536 to (-185.04, 420, -0.5) mm, rotated rx -180 ry 0 rz 90 deg; joints [-15.005, -56.613, 99.474, 158.493, 44.926, -164.412]
  MoveL 537 to (-185.04, 420, 50) mm, rotated rx -180 ry 0 rz 90 deg; joints [-15.005, -58.388, 99.177, 157.692, 43.003, -163.298]
  MoveL 538 to (-215.04, 420, 50) mm, rotated rx 180 ry 0 rz 90 deg; joints [-14.096, -58.669, 99.649, 159.048, 42.928, -164.338]
  MoveL 539 to (-215.04, 420, -0.5) mm, rotated rx -180 ry 0 rz 90 deg; joints [-14.096, -56.885, 99.947, 159.808, 44.878, -165.394]
  MoveL 540 to (-215.04, 420, 50) mm, rotated rx 180 ry 0 rz 90 deg; joints [-14.096, -58.669, 99.649, 159.048, 42.928, -164.338]
  MoveL 541 to (-260.74, 420, 50) mm, rotated rx -180 ry 0 rz 90 deg; joints [-12.698, -59.063, 100.31, 161.132, 42.821, -165.928]
  MoveL 542 to (-260.74, 420, -0.5) mm, rotated rx 180 ry 0 rz 90 deg; joints [-12.698, -57.265, 100.609, 161.826, 44.808, -166.89]
  MoveL 543 to (-260.74, 420, 50) mm, rotated rx -180 ry 0 rz 90 deg; joints [-12.698, -59.063, 100.31, 161.132, 42.821, -165.928]
  MoveL 544 to (-290.74, 420, 50) mm, rotated rx -180 ry 0 rz 90 deg; joints [-11.771, -59.299, 100.706, 162.512, 42.755, -166.974]
  MoveL 545 to (-290.74, 420, -0.5) mm, rotated rx 180 ry 0 rz 90 deg; joints [-11.771, -57.493, 101.005, 163.161, 44.766, -167.872]
  MoveL 546 to (-290.74, 420, 50) mm, rotated rx -180 ry 0 rz 90 deg; joints [-11.771, -59.299, 100.706, 162.512, 42.755, -166.974]
  MoveL 547 to (-336.44, 420, 50) mm, rotated rx -180 ry 0 rz 90 deg; joints [-10.348, -59.625, 101.249, 164.629, 42.663, -168.572]
  MoveL 548 to (-336.44, 420, -0.5) mm, rotated rx -180 ry 0 rz 90 deg; joints [-10.348, -57.808, 101.549, 165.206, 44.706, -169.369]
  MoveL 549 to (-336.44, 420, 50) mm, rotated rx -180 ry 0 rz 90 deg; joints [-10.348, -59.625, 101.249, 164.629, 42.663, -168.572]
  MoveL 550 to (-366.44, 420, 50) mm, rotated rx -180 ry 0 rz 90 deg; joints [-9.407, -59.815, 101.567, 166.029, 42.608, -169.624]
  MoveL 551 to (-366.44, 420, -0.5) mm, rotated rx -180 ry 0 rz 90 deg; joints [-9.407, -57.992, 101.867, 166.557, 44.671, -170.353]
  MoveL 552 to (-366.44, 420, 50) mm, rotated rx -180 ry 0 rz 90 deg; joints [-9.407, -59.815, 101.567, 166.029, 42.608, -169.624]
  MoveL 553 to (-33.64, 730, 50) mm, rotated rx -180 ry 0 rz 90 deg; joints [-23.192, -67.373, 113.758, 149.385, 50.65, -159.434]
  MoveL 554 to (-33.64, 730, -0.5) mm, rotated rx 180 ry 0 rz 90 deg; joints [-23.192, -65.244, 114.082, 150.357, 52.771, -161.002]
  MoveL 555 to (-33.64, 730, 50) mm, rotated rx -180 ry 0 rz 90 deg; joints [-23.192, -67.373, 113.758, 149.385, 50.65, -159.434]
  MoveL 556 to (-63.64, 730, 50) mm, rotated rx 180 ry 0 rz 90 deg; joints [-22.191, -67.798, 114.418, 150.698, 50.509, -160.358]
  MoveL 557 to (-63.64, 730, -0.5) mm, rotated rx 180 ry 0 rz 90 deg; joints [-22.191, -65.65, 114.744, 151.644, 52.677, -161.88]
  MoveL 558 to (-63.64, 730, 50) mm, rotated rx 180 ry 0 rz 90 deg; joints [-22.191, -67.798, 114.418, 150.698, 50.509, -160.358]
  MoveL 559 to (-109.34, 730, 50) mm, rotated rx -180 ry 0 rz 90 deg; joints [-20.639, -68.413, 115.366, 152.734, 50.298, -161.777]
  MoveL 560 to (-109.34, 730, -0.5) mm, rotated rx 180 ry 0 rz 90 deg; joints [-20.639, -66.235, 115.694, 153.636, 52.535, -163.223]
  MoveL 561 to (-109.34, 730, 50) mm, rotated rx -180 ry 0 rz 90 deg; joints [-20.639, -68.413, 115.366, 152.734, 50.298, -161.777]
  MoveL 562 to (-139.34, 730, 50) mm, rotated rx 180 ry 0 rz 90 deg; joints [-19.602, -68.793, 115.949, 154.093, 50.163, -162.716]
  MoveL 563 to (-139.34, 730, -0.5) mm, rotated rx 180 ry 0 rz 90 deg; joints [-19.602, -66.597, 116.279, 154.964, 52.445, -164.109]
  MoveL 564 to (-139.34, 730, 50) mm, rotated rx 180 ry 0 rz 90 deg; joints [-19.602, -68.793, 115.949, 154.093, 50.163, -162.716]
  MoveL 565 to (-185.04, 730, 50) mm, rotated rx -180 ry 0 rz 90 deg; joints [-17.997, -69.337, 116.778, 156.2, 49.965, -164.161]
  MoveL 566 to (-185.04, 730, -0.5) mm, rotated rx -180 ry 0 rz 90 deg; joints [-17.997, -67.114, 117.111, 157.018, 52.311, -165.464]
  MoveL 567 to (-185.04, 730, 50) mm, rotated rx -180 ry 0 rz 90 deg; joints [-17.997, -69.337, 116.778, 156.2, 49.965, -164.161]
  MoveL 568 to (-215.04, 730, 50) mm, rotated rx -180 ry 0 rz 90 deg; joints [-16.928, -69.671, 117.283, 157.605, 49.84, -165.118]
  MoveL 569 to (-215.04, 730, -0.5) mm, rotated rx -180 ry 0 rz 90 deg; joints [-16.928, -67.43, 117.618, 158.386, 52.227, -166.358]
  MoveL 570 to (-215.04, 730, 50) mm, rotated rx -180 ry 0 rz 90 deg; joints [-16.928, -69.671, 117.283, 157.605, 49.84, -165.118]
  MoveL 571 to (-260.74, 730, 50) mm, rotated rx -180 ry 0 rz 90 deg; joints [-15.275, -70.14, 117.992, 159.779, 49.658, -166.589]
  MoveL 572 to (-260.74, 730, -0.5) mm, rotated rx 180 ry 0 rz 90 deg; joints [-15.275, -67.876, 118.329, 160.498, 52.105, -167.728]
  MoveL 573 to (-260.74, 730, 50) mm, rotated rx -180 ry 0 rz 90 deg; joints [-15.275, -70.14, 117.992, 159.779, 49.658, -166.589]
  MoveL 574 to (-290.74, 730, 50) mm, rotated rx 180 ry 0 rz 90 deg; joints [-14.175, -70.424, 118.417, 161.227, 49.546, -167.563]
  MoveL 575 to (-290.74, 730, -0.5) mm, rotated rx 180 ry 0 rz 90 deg; joints [-14.175, -68.145, 118.756, 161.902, 52.029, -168.631]
  MoveL 576 to (-290.74, 730, 50) mm, rotated rx 180 ry 0 rz 90 deg; joints [-14.175, -70.424, 118.417, 161.227, 49.546, -167.563]
  MoveL 577 to (-336.44, 730, 50) mm, rotated rx 180 ry 0 rz 90 deg; joints [-12.479, -70.815, 119.003, 163.462, 49.387, -169.06]
  MoveL 578 to (-336.44, 730, -0.5) mm, rotated rx -180 ry 0 rz 90 deg; joints [-12.479, -68.516, 119.344, 164.067, 51.922, -170.015]
  MoveL 579 to (-336.44, 730, 50) mm, rotated rx 180 ry 0 rz 90 deg; joints [-12.479, -70.815, 119.003, 163.462, 49.387, -169.06]
  MoveL 580 to (-366.44, 730, 50) mm, rotated rx 180 ry 0 rz 90 deg; joints [-11.354, -71.046, 119.347, 164.948, 49.292, -170.052]
  MoveL 581 to (-366.44, 730, -0.5) mm, rotated rx 180 ry 0 rz 90 deg; joints [-11.354, -68.735, 119.689, 165.504, 51.858, -170.928]
  MoveL 582 to (-366.44, 730, 50) mm, rotated rx 180 ry 0 rz 90 deg; joints [-11.354, -71.046, 119.347, 164.948, 49.292, -170.052]
  MoveL 583 to (-33.64, 1020, 50) mm, rotated rx 180 ry 0 rz 90 deg; joints [-28.122, -77.24, 128.147, 145.449, 56.211, -159.045]
  MoveL 584 to (-33.64, 1020, -0.5) mm, rotated rx -180 ry 0 rz 90 deg; joints [-28.122, -74.558, 128.529, 146.542, 58.751, -161.078]
  MoveL 585 to (-33.64, 1020, 50) mm, rotated rx 180 ry 0 rz 90 deg; joints [-28.122, -77.24, 128.147, 145.449, 56.211, -159.045]
  MoveL 586 to (-63.64, 1020, 50) mm, rotated rx -180 ry 0 rz 90 deg; joints [-26.969, -77.787, 128.882, 146.82, 55.963, -159.897]
  MoveL 587 to (-63.64, 1020, -0.5) mm, rotated rx -180 ry 0 rz 90 deg; joints [-26.969, -75.068, 129.269, 147.897, 58.578, -161.889]
  MoveL 588 to (-63.64, 1020, 50) mm, rotated rx -180 ry 0 rz 90 deg; joints [-26.969, -77.787, 128.882, 146.82, 55.963, -159.897]
  MoveL 589 to (-109.34, 1020, 50) mm, rotated rx 180 ry 0 rz 90 deg; joints [-25.166, -78.587, 129.943, 148.971, 55.584, -161.222]
  MoveL 590 to (-109.34, 1020, -0.5) mm, rotated rx -180 ry 0 rz 90 deg; joints [-25.166, -75.812, 130.336, 150.017, 58.313, -163.14]
  MoveL 591 to (-109.34, 1020, 50) mm, rotated rx 180 ry 0 rz 90 deg; joints [-25.166, -78.587, 129.943, 148.971, 55.584, -161.222]
  MoveL 592 to (-139.34, 1020, 50) mm, rotated rx 180 ry 0 rz 90 deg; joints [-23.953, -79.087, 130.599, 150.423, 55.337, -162.11]
  MoveL 593 to (-139.34, 1020, -0.5) mm, rotated rx -180 ry 0 rz 90 deg; joints [-23.953, -76.277, 130.996, 151.445, 58.14, -163.973]
  MoveL 594 to (-139.34, 1020, 50) mm, rotated rx 180 ry 0 rz 90 deg; joints [-23.953, -79.087, 130.599, 150.423, 55.337, -162.11]
  MoveL 595 to (-185.04, 1020, 50) mm, rotated rx 180 ry 0 rz 90 deg; joints [-22.061, -79.81, 131.535, 152.697, 54.965, -163.493]
  MoveL 596 to (-185.04, 1020, -0.5) mm, rotated rx -180 ry 0 rz 90 deg; joints [-22.061, -76.948, 131.939, 153.675, 57.879, -165.261]
  MoveL 597 to (-185.04, 1020, 50) mm, rotated rx 180 ry 0 rz 90 deg; joints [-22.061, -79.81, 131.535, 152.697, 54.965, -163.493]
  MoveL 598 to (-215.04, 1020, 50) mm, rotated rx -180 ry 0 rz 90 deg; joints [-20.79, -80.257, 132.108, 154.23, 54.726, -164.422]
  MoveL 599 to (-215.04, 1020, -0.5) mm, rotated rx -180 ry 0 rz 90 deg; joints [-20.79, -77.362, 132.515, 155.174, 57.711, -166.119]
  MoveL 600 to (-215.04, 1020, 50) mm, rotated rx -180 ry 0 rz 90 deg; joints [-20.79, -80.257, 132.108, 154.23, 54.726, -164.422]
  MoveL 601 to (-260.74, 1020, 50) mm, rotated rx 180 ry 0 rz 90 deg; joints [-18.812, -80.894, 132.914, 156.626, 54.373, -165.869]
  MoveL 602 to (-260.74, 1020, -0.5) mm, rotated rx -180 ry 0 rz 90 deg; joints [-18.812, -77.952, 133.327, 157.511, 57.463, -167.447]
  MoveL 603 to (-260.74, 1020, 50) mm, rotated rx 180 ry 0 rz 90 deg; joints [-18.812, -80.894, 132.914, 156.626, 54.373, -165.869]
  MoveL 604 to (-290.74, 1020, 50) mm, rotated rx -180 ry 0 rz 90 deg; joints [-17.488, -81.282, 133.4, 158.239, 54.151, -166.842]
  MoveL 605 to (-290.74, 1020, -0.5) mm, rotated rx 180 ry 0 rz 90 deg; joints [-17.488, -78.31, 133.816, 159.079, 57.307, -168.333]
  MoveL 606 to (-290.74, 1020, 50) mm, rotated rx -180 ry 0 rz 90 deg; joints [-17.488, -81.282, 133.4, 158.239, 54.151, -166.842]
  MoveL 607 to (-336.44, 1020, 50) mm, rotated rx 180 ry 0 rz 90 deg; joints [-15.434, -81.823, 134.071, 160.753, 53.831, -168.356]
  MoveL 608 to (-336.44, 1020, -0.5) mm, rotated rx 180 ry 0 rz 90 deg; joints [-15.434, -78.809, 134.493, 161.517, 57.082, -169.705]
  MoveL 609 to (-336.44, 1020, 50) mm, rotated rx 180 ry 0 rz 90 deg; joints [-15.434, -81.823, 134.071, 160.753, 53.831, -168.356]
  MoveL 610 to (-366.44, 1020, 50) mm, rotated rx -180 ry 0 rz 90 deg; joints [-14.062, -82.144, 134.466, 162.439, 53.636, -169.372]
  MoveL 611 to (-366.44, 1020, -0.5) mm, rotated rx -180 ry 0 rz 90 deg; joints [-14.062, -79.106, 134.891, 163.148, 56.945, -170.619]
  MoveL 612 to (-366.44, 1020, 50) mm, rotated rx -180 ry 0 rz 90 deg; joints [-14.062, -82.144, 134.466, 162.439, 53.636, -169.372]
  MoveL 613 to (-450, 50, 50) mm, rotated rx 180 ry 0 rz 90 deg; joints [-5.599, -45.905, 77.379, 169.365, 31.918, -170.944]
  MoveL 614 to (-450, 50, -0.5) mm, rotated rx -180 ry 0 rz 90 deg; joints [-5.599, -44.463, 77.676, 169.852, 33.629, -171.524]
  MoveL 615 to (-450, 50, 50) mm, rotated rx 180 ry 0 rz 90 deg; joints [-5.599, -45.905, 77.379, 169.365, 31.918, -170.944]
  MoveL 616 to (-450, 100, 50) mm, rotated rx 180 ry 0 rz 90 deg; joints [-5.732, -47.978, 81.093, 169.588, 33.552, -171.294]
  MoveL 617 to (-450, 100, -0.5) mm, rotated rx -180 ry 0 rz 90 deg; joints [-5.732, -46.49, 81.387, 170.048, 35.305, -171.851]
  MoveL 618 to (-450, 100, 50) mm, rotated rx 180 ry 0 rz 90 deg; joints [-5.732, -47.978, 81.093, 169.588, 33.552, -171.294]
  MoveL 619 to (-450, 150, 50) mm, rotated rx -180 ry 0 rz 90 deg; joints [-5.872, -49.995, 84.675, 169.755, 35.111, -171.589]
  MoveL 620 to (-450, 150, -0.5) mm, rotated rx 180 ry 0 rz 90 deg; joints [-5.872, -48.46, 84.967, 170.193, 36.911, -172.131]
  MoveL 621 to (-450, 150, 50) mm, rotated rx -180 ry 0 rz 90 deg; joints [-5.872, -49.995, 84.675, 169.755, 35.111, -171.589]
  MoveL 622 to (-450, 200, 50) mm, rotated rx -180 ry 0 rz 90 deg; joints [-6.018, -51.965, 88.139, 169.873, 36.603, -171.84]
  MoveL 623 to (-450, 200, -0.5) mm, rotated rx 180 ry 0 rz 90 deg; joints [-6.018, -50.379, 88.431, 170.294, 38.453, -172.371]
  MoveL 624 to (-450, 200, 50) mm, rotated rx -180 ry 0 rz 90 deg; joints [-6.018, -51.965, 88.139, 169.873, 36.603, -171.84]
  MoveL 625 to (-450, 250, 50) mm, rotated rx -180 ry 0 rz 90 deg; joints [-6.172, -53.895, 91.5, 169.951, 38.034, -172.054]
  MoveL 626 to (-450, 250, -0.5) mm, rotated rx -180 ry 0 rz 90 deg; joints [-6.172, -52.257, 91.792, 170.359, 39.936, -172.579]
  MoveL 627 to (-450, 250, 50) mm, rotated rx -180 ry 0 rz 90 deg; joints [-6.172, -53.895, 91.5, 169.951, 38.034, -172.054]
  MoveL 628 to (-450, 300, 50) mm, rotated rx 180 ry 0 rz 90 deg; joints [-6.334, -55.793, 94.769, 169.992, 39.406, -172.236]
  MoveL 629 to (-450, 300, -0.5) mm, rotated rx 180 ry 0 rz 90 deg; joints [-6.334, -54.1, 95.062, 170.39, 41.364, -172.758]
  MoveL 630 to (-450, 300, 50) mm, rotated rx 180 ry 0 rz 90 deg; joints [-6.334, -55.793, 94.769, 169.992, 39.406, -172.236]
  MoveL 631 to (-450, 350, 50) mm, rotated rx 180 ry 0 rz 90 deg; joints [-6.504, -57.664, 97.955, 170.001, 40.723, -172.39]
  MoveL 632 to (-450, 350, -0.5) mm, rotated rx -180 ry 0 rz 90 deg; joints [-6.504, -55.913, 98.251, 170.392, 42.741, -172.913]
  MoveL 633 to (-450, 350, 50) mm, rotated rx 180 ry 0 rz 90 deg; joints [-6.504, -57.664, 97.955, 170.001, 40.723, -172.39]
  MoveL 634 to (-450, 400, 50) mm, rotated rx -180 ry 0 rz 90 deg; joints [-6.684, -59.515, 101.065, 169.981, 41.988, -172.519]
  MoveL 635 to (-450, 400, -0.5) mm, rotated rx 180 ry 0 rz 90 deg; joints [-6.684, -57.701, 101.365, 170.367, 44.07, -173.047]
  MoveL 636 to (-450, 400, 50) mm, rotated rx -180 ry 0 rz 90 deg; joints [-6.684, -59.515, 101.065, 169.981, 41.988, -172.519]
  MoveL 637 to (-450, 450, 50) mm, rotated rx -180 ry 0 rz 90 deg; joints [-6.874, -61.35, 104.108, 169.931, 43.202, -172.625]
  MoveL 638 to (-450, 450, -0.5) mm, rotated rx -180 ry 0 rz 90 deg; joints [-6.874, -59.471, 104.412, 170.315, 45.352, -173.161]
  MoveL 639 to (-450, 450, 50) mm, rotated rx -180 ry 0 rz 90 deg; joints [-6.874, -61.35, 104.108, 169.931, 43.202, -172.625]
  MoveL 640 to (-450, 500, 50) mm, rotated rx 180 ry 0 rz 90 deg; joints [-7.075, -63.174, 107.089, 169.855, 44.366, -172.71]
  MoveL 641 to (-450, 500, -0.5) mm, rotated rx -180 ry 0 rz 90 deg; joints [-7.075, -61.226, 107.398, 170.238, 46.589, -173.257]
  MoveL 642 to (-450, 500, 50) mm, rotated rx 180 ry 0 rz 90 deg; joints [-7.075, -63.174, 107.089, 169.855, 44.366, -172.71]
  MoveL 643 to (-450, 550, 50) mm, rotated rx -180 ry 0 rz 90 deg; joints [-7.288, -64.993, 110.013, 169.751, 45.48, -172.775]
  MoveL 644 to (-450, 550, -0.5) mm, rotated rx 180 ry 0 rz 90 deg; joints [-7.288, -62.97, 110.327, 170.137, 47.782, -173.336]
  MoveL 645 to (-450, 550, 50) mm, rotated rx -180 ry 0 rz 90 deg; joints [-7.288, -64.993, 110.013, 169.751, 45.48, -172.775]
  MoveL 646 to (-450, 600, 50) mm, rotated rx 180 ry 0 rz 90 deg; joints [-7.514, -66.812, 112.884, 169.621, 46.544, -172.82]
  MoveL 647 to (-450, 600, -0.5) mm, rotated rx -180 ry 0 rz 90 deg; joints [-7.514, -64.709, 113.206, 170.011, 48.931, -173.399]
  MoveL 648 to (-450, 600, 50) mm, rotated rx 180 ry 0 rz 90 deg; joints [-7.514, -66.812, 112.884, 169.621, 46.544, -172.82]
  MoveL 649 to (-450, 650, 50) mm, rotated rx 180 ry 0 rz 90 deg; joints [-7.755, -68.635, 115.707, 169.464, 47.557, -172.846]
  MoveL 650 to (-450, 650, -0.5) mm, rotated rx -180 ry 0 rz 90 deg; joints [-7.755, -66.446, 116.036, 169.859, 50.035, -173.446]
  MoveL 651 to (-450, 650, 50) mm, rotated rx 180 ry 0 rz 90 deg; joints [-7.755, -68.635, 115.707, 169.464, 47.557, -172.846]
  MoveL 652 to (-450, 700, 50) mm, rotated rx 180 ry 0 rz 90 deg; joints [-8.012, -70.468, 118.484, 169.278, 48.517, -172.851]
  MoveL 653 to (-450, 700, -0.5) mm, rotated rx -180 ry 0 rz 90 deg; joints [-8.012, -68.187, 118.823, 169.682, 51.093, -173.477]
  MoveL 654 to (-450, 700, 50) mm, rotated rx 180 ry 0 rz 90 deg; joints [-8.012, -70.468, 118.484, 169.278, 48.517, -172.851]
  MoveL 655 to (-450, 750, 50) mm, rotated rx -180 ry 0 rz 90 deg; joints [-8.286, -72.317, 121.22, 169.063, 49.423, -172.835]
  MoveL 656 to (-450, 750, -0.5) mm, rotated rx 180 ry 0 rz 90 deg; joints [-8.286, -69.936, 121.569, 169.478, 52.105, -173.492]
  MoveL 657 to (-450, 750, 50) mm, rotated rx -180 ry 0 rz 90 deg; joints [-8.286, -72.317, 121.22, 169.063, 49.423, -172.835]
  MoveL 658 to (-450, 800, 50) mm, rotated rx 180 ry 0 rz 90 deg; joints [-8.579, -74.189, 123.917, 168.815, 50.269, -172.797]
  MoveL 659 to (-450, 800, -0.5) mm, rotated rx 180 ry 0 rz 90 deg; joints [-8.579, -71.699, 124.278, 169.244, 53.067, -173.488]
  MoveL 660 to (-450, 800, 50) mm, rotated rx 180 ry 0 rz 90 deg; joints [-8.579, -74.189, 123.917, 168.815, 50.269, -172.797]
  MoveL 661 to (-450, 850, 50) mm, rotated rx -180 ry 0 rz 90 deg; joints [-8.894, -76.089, 126.577, 168.534, 51.054, -172.734]
  MoveL 662 to (-450, 850, -0.5) mm, rotated rx 180 ry 0 rz 90 deg; joints [-8.894, -73.482, 126.951, 168.98, 53.977, -173.466]
  MoveL 663 to (-450, 850, 50) mm, rotated rx -180 ry 0 rz 90 deg; joints [-8.894, -76.089, 126.577, 168.534, 51.054, -172.734]
  MoveL 664 to (-450, 900, 50) mm, rotated rx 180 ry 0 rz 90 deg; joints [-9.232, -78.027, 129.202, 168.215, 51.77, -172.643]
  MoveL 665 to (-450, 900, -0.5) mm, rotated rx -180 ry 0 rz 90 deg; joints [-9.232, -75.292, 129.591, 168.682, 54.831, -173.424]
  MoveL 666 to (-450, 900, 50) mm, rotated rx 180 ry 0 rz 90 deg; joints [-9.232, -78.027, 129.202, 168.215, 51.77, -172.643]
  MoveL 667 to (-450, 950, 50) mm, rotated rx 180 ry 0 rz 90 deg; joints [-9.597, -80.012, 131.794, 167.855, 52.411, -172.521]
  MoveL 668 to (-450, 950, -0.5) mm, rotated rx -180 ry 0 rz 90 deg; joints [-9.597, -77.135, 132.199, 168.346, 55.622, -173.357]
  MoveL 669 to (-450, 950, 50) mm, rotated rx 180 ry 0 rz 90 deg; joints [-9.597, -80.012, 131.794, 167.855, 52.411, -172.521]
  MoveL 670 to (-450, 1000, 50) mm, rotated rx 180 ry 0 rz 90 deg; joints [-9.992, -82.053, 134.355, 167.447, 52.97, -172.363]
  MoveL 671 to (-450, 1000, -0.5) mm, rotated rx 180 ry 0 rz 90 deg; joints [-9.992, -79.022, 134.779, 167.969, 56.346, -173.264]
  MoveL 672 to (-450, 1000, 50) mm, rotated rx 180 ry 0 rz 90 deg; joints [-9.992, -82.053, 134.355, 167.447, 52.97, -172.363]
  MoveL 673 to (-450, 1050, 50) mm, rotated rx -180 ry 0 rz 90 deg; joints [-10.42, -84.166, 136.885, 166.987, 53.435, -172.161]
  MoveL 674 to (-450, 1050, -0.5) mm, rotated rx 180 ry 0 rz 90 deg; joints [-10.42, -80.963, 137.33, 167.546, 56.993, -173.14]
  MoveL 675 to (-450, 1050, 50) mm, rotated rx -180 ry 0 rz 90 deg; joints [-10.42, -84.166, 136.885, 166.987, 53.435, -172.161]
  MoveL 676 to (-450, 1100, 50) mm, rotated rx -180 ry 0 rz 90 deg; joints [-10.886, -86.364, 139.385, 166.465, 53.793, -171.907]
  MoveL 677 to (-450, 1100, -0.5) mm, rotated rx -180 ry 0 rz 90 deg; joints [-10.886, -82.972, 139.854, 167.069, 57.552, -172.977]
  MoveL 678 to (-450, 1100, 50) mm, rotated rx -180 ry 0 rz 90 deg; joints [-10.886, -86.364, 139.385, 166.465, 53.793, -171.907]
  MoveL 679 to (-450, 1150, 50) mm, rotated rx -180 ry 0 rz 90 deg; joints [-11.395, -88.668, 141.855, 165.871, 54.028, -171.589]
  MoveL 680 to (-450, 1150, -0.5) mm, rotated rx -180 ry 0 rz 90 deg; joints [-11.395, -85.064, 142.352, 166.53, 58.011, -172.768]
  MoveL 681 to (-450, 1150, 50) mm, rotated rx -180 ry 0 rz 90 deg; joints [-11.395, -88.668, 141.855, 165.871, 54.028, -171.589]
  MoveL 682 to (-450, 1200, 50) mm, rotated rx -180 ry 0 rz 90 deg; joints [-11.953, -91.1, 144.296, 165.19, 54.12, -171.192]
  MoveL 683 to (-450, 1200, -0.5) mm, rotated rx 180 ry 0 rz 90 deg; joints [-11.953, -87.26, 144.825, 165.919, 58.351, -172.502]
  MoveL 684 to (-450, 1200, 50) mm, rotated rx -180 ry 0 rz 90 deg; joints [-11.953, -91.1, 144.296, 165.19, 54.12, -171.192]
  MoveL 685 to (-450, 1250, 50) mm, rotated rx 180 ry 0 rz 90 deg; joints [-12.567, -93.692, 146.707, 164.406, 54.042, -170.693]
  MoveL 686 to (-450, 1250, -0.5) mm, rotated rx -180 ry 0 rz 90 deg; joints [-12.567, -89.587, 147.272, 165.223, 58.55, -172.164]
  MoveL 687 to (-450, 1250, 50) mm, rotated rx 180 ry 0 rz 90 deg; joints [-12.567, -93.692, 146.707, 164.406, 54.042, -170.693]
  MoveL 688 to (-450, 1300, 50) mm, rotated rx 180 ry 0 rz 90 deg; joints [-13.248, -96.482, 149.086, 163.494, 53.761, -170.064]
  MoveL 689 to (-450, 1300, -0.5) mm, rotated rx -180 ry 0 rz 90 deg; joints [-13.248, -92.077, 149.694, 164.423, 58.579, -171.731]
  MoveL 690 to (-450, 1300, 50) mm, rotated rx 180 ry 0 rz 90 deg; joints [-13.248, -96.482, 149.086, 163.494, 53.761, -170.064]
  MoveL 691 to (-450, 1350, 50) mm, rotated rx -180 ry 0 rz 90 deg; joints [-14.004, -99.519, 151.431, 162.417, 53.234, -169.26]
  MoveL 692 to (-450, 1350, -0.5) mm, rotated rx -180 ry 0 rz 90 deg; joints [-14.004, -94.776, 152.09, 163.494, 58.4, -171.174]
  MoveL 693 to (-450, 1350, 50) mm, rotated rx -180 ry 0 rz 90 deg; joints [-14.004, -99.519, 151.431, 162.417, 53.234, -169.26]
  MoveL 694 to (-450, 1400, 50) mm, rotated rx -180 ry 0 rz 90 deg; joints [-14.85, -102.871, 153.738, 161.128, 52.408, -168.221]
  MoveL 695 to (-450, 1400, -0.5) mm, rotated rx 180 ry 0 rz 90 deg; joints [-14.85, -97.745, 154.457, 162.401, 57.96, -170.448]
  MoveL 696 to (-450, 1400, 50) mm, rotated rx -180 ry 0 rz 90 deg; joints [-14.85, -102.871, 153.738, 161.128, 52.408, -168.221]
  MoveL 697 to (-450, 1450, 50) mm, rotated rx 180 ry 0 rz 70 deg; joints [-22.417, -102.648, 153.594, 130.362, 62.281, -151.309]
  MoveL 698 to (-450, 1450, -0.5) mm, rotated rx -180 ry 0 rz 70 deg; joints [-22.417, -97.548, 154.308, 132.471, 66.13, -156.151]
  MoveL 699 to (-450, 1450, 50) mm, rotated rx 180 ry 0 rz 70 deg; joints [-22.417, -102.648, 153.594, 130.362, 62.281, -151.309]
  MoveL 700 to (-578.4, 50, 50) mm, rotated rx 180 ry 0 rz 90 deg; joints [-2.182, -46.273, 78.04, 175.861, 31.835, -176.482]
  MoveL 701 to (-578.4, 50, -0.5) mm, rotated rx 180 ry 0 rz 90 deg; joints [-2.182, -44.822, 78.336, 176.053, 33.576, -176.71]
  MoveL 702 to (-578.4, 50, 50) mm, rotated rx -180 ry 0 rz 90 deg; joints [-2.182, -46.273, 78.04, 175.861, 31.835, -176.482]
  MoveL 703 to (-578.4, 100, 50) mm, rotated rx -180 ry 0 rz 90 deg; joints [-2.234, -48.344, 81.745, 175.947, 33.467, -176.617]
  MoveL 704 to (-578.4, 100, -0.5) mm, rotated rx 180 ry 0 rz 90 deg; joints [-2.234, -46.848, 82.038, 176.128, 35.252, -176.836]
  MoveL 705 to (-578.4, 100, 50) mm, rotated rx -180 ry 0 rz 90 deg; joints [-2.234, -48.344, 81.745, 175.947, 33.467, -176.617]
  MoveL 706 to (-578.4, 150, 50) mm, rotated rx 180 ry 0 rz 90 deg; joints [-2.288, -50.361, 85.32, 176.011, 35.024, -176.731]
  MoveL 707 to (-578.4, 150, -0.5) mm, rotated rx -180 ry 0 rz 90 deg; joints [-2.288, -48.816, 85.611, 176.183, 36.857, -176.944]
  MoveL 708 to (-578.4, 150, 50) mm, rotated rx 180 ry 0 rz 90 deg; joints [-2.288, -50.361, 85.32, 176.011, 35.024, -176.731]
  MoveL 709 to (-578.4, 200, 50) mm, rotated rx 180 ry 0 rz 90 deg; joints [-2.346, -52.332, 88.78, 176.056, 36.513, -176.828]
  MoveL 710 to (-578.4, 200, -0.5) mm, rotated rx 180 ry 0 rz 90 deg; joints [-2.346, -50.736, 89.071, 176.222, 38.396, -177.037]
  MoveL 711 to (-578.4, 200, 50) mm, rotated rx 180 ry 0 rz 90 deg; joints [-2.346, -52.332, 88.78, 176.056, 36.513, -176.828]
  MoveL 712 to (-578.4, 250, 50) mm, rotated rx 180 ry 0 rz 90 deg; joints [-2.406, -54.264, 92.139, 176.085, 37.939, -176.91]
  MoveL 713 to (-578.4, 250, -0.5) mm, rotated rx 180 ry 0 rz 90 deg; joints [-2.406, -52.616, 92.431, 176.246, 39.876, -177.117]
  MoveL 714 to (-578.4, 250, 50) mm, rotated rx 180 ry 0 rz 90 deg; joints [-2.406, -54.264, 92.139, 176.085, 37.939, -176.91]
  MoveL 715 to (-578.4, 300, 50) mm, rotated rx 180 ry 0 rz 90 deg; joints [-2.47, -56.166, 95.407, 176.1, 39.306, -176.98]
  MoveL 716 to (-578.4, 300, -0.5) mm, rotated rx -180 ry 0 rz 90 deg; joints [-2.47, -54.462, 95.701, 176.257, 41.3, -177.186]
  MoveL 717 to (-578.4, 300, 50) mm, rotated rx 180 ry 0 rz 90 deg; joints [-2.47, -56.166, 95.407, 176.1, 39.306, -176.98]
  MoveL 718 to (-578.4, 350, 50) mm, rotated rx 180 ry 0 rz 90 deg; joints [-2.537, -58.043, 98.594, 176.102, 40.617, -177.039]
  MoveL 719 to (-578.4, 350, -0.5) mm, rotated rx 180 ry 0 rz 90 deg; joints [-2.537, -56.279, 98.891, 176.256, 42.673, -177.246]
  MoveL 720 to (-578.4, 350, 50) mm, rotated rx 180 ry 0 rz 90 deg; joints [-2.537, -58.043, 98.594, 176.102, 40.617, -177.039]
  MoveL 721 to (-578.4, 400, 50) mm, rotated rx 180 ry 0 rz 90 deg; joints [-2.607, -59.9, 101.708, 176.092, 41.874, -177.088]
  MoveL 722 to (-578.4, 400, -0.5) mm, rotated rx -180 ry 0 rz 90 deg; joints [-2.607, -58.074, 102.009, 176.245, 43.997, -177.297]
  MoveL 723 to (-578.4, 400, 50) mm, rotated rx 180 ry 0 rz 90 deg; joints [-2.607, -59.9, 101.708, 176.092, 41.874, -177.088]
  MoveL 724 to (-578.4, 450, 50) mm, rotated rx -180 ry 0 rz 90 deg; joints [-2.682, -61.744, 104.756, 176.072, 43.079, -177.129]
  MoveL 725 to (-578.4, 450, -0.5) mm, rotated rx -180 ry 0 rz 90 deg; joints [-2.682, -59.85, 105.061, 176.224, 45.273, -177.341]
  MoveL 726 to (-578.4, 450, 50) mm, rotated rx -180 ry 0 rz 90 deg; joints [-2.682, -61.744, 104.756, 176.072, 43.079, -177.129]
  MoveL 727 to (-578.4, 500, 50) mm, rotated rx -180 ry 0 rz 90 deg; joints [-2.761, -63.578, 107.743, 176.04, 44.233, -177.161]
  MoveL 728 to (-578.4, 500, -0.5) mm, rotated rx -180 ry 0 rz 90 deg; joints [-2.761, -61.614, 108.053, 176.192, 46.502, -177.377]
  MoveL 729 to (-578.4, 500, 50) mm, rotated rx -180 ry 0 rz 90 deg; joints [-2.761, -63.578, 107.743, 176.04, 44.233, -177.161]
  MoveL 730 to (-578.4, 550, 50) mm, rotated rx -180 ry 0 rz 90 deg; joints [-2.845, -65.409, 110.674, 175.998, 45.335, -177.185]
  MoveL 731 to (-578.4, 550, -0.5) mm, rotated rx -180 ry 0 rz 90 deg; joints [-2.845, -63.368, 110.99, 176.151, 47.686, -177.407]
  MoveL 732 to (-578.4, 550, 50) mm, rotated rx -180 ry 0 rz 90 deg; joints [-2.845, -65.409, 110.674, 175.998, 45.335, -177.185]
  MoveL 733 to (-578.4, 600, 50) mm, rotated rx 180 ry 0 rz 90 deg; joints [-2.934, -67.242, 113.554, 175.946, 46.385, -177.201]
  MoveL 734 to (-578.4, 600, -0.5) mm, rotated rx 180 ry 0 rz 90 deg; joints [-2.934, -65.119, 113.878, 176.1, 48.825, -177.43]
  MoveL 735 to (-578.4, 600, 50) mm, rotated rx 180 ry 0 rz 90 deg; joints [-2.934, -67.242, 113.554, 175.946, 46.385, -177.201]
  MoveL 736 to (-578.4, 650, 50) mm, rotated rx 180 ry 0 rz 90 deg; joints [-3.029, -69.081, 116.388, 175.882, 47.381, -177.209]
  MoveL 737 to (-578.4, 650, -0.5) mm, rotated rx 180 ry 0 rz 90 deg; joints [-3.029, -66.87, 116.72, 176.04, 49.917, -177.448]
  MoveL 738 to (-578.4, 650, 50) mm, rotated rx 180 ry 0 rz 90 deg; joints [-3.029, -69.081, 116.388, 175.882, 47.381, -177.209]
  MoveL 739 to (-578.4, 700, 50) mm, rotated rx 180 ry 0 rz 90 deg; joints [-3.13, -70.933, 119.178, 175.807, 48.321, -177.209]
  MoveL 740 to (-578.4, 700, -0.5) mm, rotated rx 180 ry 0 rz 90 deg; joints [-3.13, -68.627, 119.519, 175.968, 50.961, -177.458]
  MoveL 741 to (-578.4, 700, 50) mm, rotated rx 180 ry 0 rz 90 deg; joints [-3.13, -70.933, 119.178, 175.807, 48.321, -177.209]
  MoveL 742 to (-578.4, 750, 50) mm, rotated rx 180 ry 0 rz 90 deg; joints [-3.239, -72.803, 121.927, 175.72, 49.203, -177.201]
  MoveL 743 to (-578.4, 750, -0.5) mm, rotated rx 180 ry 0 rz 90 deg; joints [-3.239, -70.395, 122.279, 175.886, 51.956, -177.462]
  MoveL 744 to (-578.4, 750, 50) mm, rotated rx 180 ry 0 rz 90 deg; joints [-3.239, -72.803, 121.927, 175.72, 49.203, -177.201]
  MoveL 745 to (-578.4, 800, 50) mm, rotated rx -180 ry 0 rz 90 deg; joints [-3.355, -74.699, 124.64, 175.62, 50.023, -177.183]
  MoveL 746 to (-578.4, 800, -0.5) mm, rotated rx 180 ry 0 rz 90 deg; joints [-3.355, -72.179, 125.004, 175.792, 52.899, -177.459]
  MoveL 747 to (-578.4, 800, 50) mm, rotated rx -180 ry 0 rz 90 deg; joints [-3.355, -74.699, 124.64, 175.62, 50.023, -177.183]
  MoveL 748 to (-578.4, 850, 50) mm, rotated rx 180 ry 0 rz 90 deg; joints [-3.48, -76.629, 127.317, 175.506, 50.775, -177.155]
  MoveL 749 to (-578.4, 850, -0.5) mm, rotated rx 180 ry 0 rz 90 deg; joints [-3.48, -73.987, 127.694, 175.686, 53.785, -177.448]
  MoveL 750 to (-578.4, 850, 50) mm, rotated rx 180 ry 0 rz 90 deg; joints [-3.48, -76.629, 127.317, 175.506, 50.775, -177.155]
  MoveL 751 to (-578.4, 900, 50) mm, rotated rx 180 ry 0 rz 90 deg; joints [-3.614, -78.6, 129.961, 175.377, 51.452, -177.115]
  MoveL 752 to (-578.4, 900, -0.5) mm, rotated rx -180 ry 0 rz 90 deg; joints [-3.614, -75.825, 130.354, 175.566, 54.61, -177.428]
  MoveL 753 to (-578.4, 900, 50) mm, rotated rx 180 ry 0 rz 90 deg; joints [-3.614, -78.6, 129.961, 175.377, 51.452, -177.115]
  MoveL 754 to (-578.4, 950, 50) mm, rotated rx -180 ry 0 rz 90 deg; joints [-3.759, -80.624, 132.574, 175.231, 52.046, -177.063]
  MoveL 755 to (-578.4, 950, -0.5) mm, rotated rx 180 ry 0 rz 90 deg; joints [-3.759, -77.702, 132.985, 175.43, 55.368, -177.399]
